LIN {X 0,Y 306.1,Z 708.373,A -85,B 0,C 180,E1 -15814.137,E2 -15814.137} C_VEL
LIN {X 0,Y 305.389,Z 716.212,A -85,B 0,C 180,E1 -15815.891,E2 -15815.891} C_VEL
LIN {X 0,Y 304.781,Z 723.046,A -85,B 0,C 180,E1 -15817.778,E2 -15817.778} C_VEL
LIN {X 0,Y 304.281,Z 728.72,A -85,B 0,C 180,E1 -15819.73,E2 -15819.73} C_VEL
LIN {X 0,Y 303.968,Z 733.701,A -85,B 0,C 180,E1 -15821.947,E2 -15821.947} C_VEL
LIN {X 0,Y 303.7,Z 736.898,A -85,B 0,C 180,E1 -15823.878,E2 -15823.878} C_VEL
LIN {X 0,Y 303.693,Z 738.582,A -85,B 0,C 180,E1 -15825.253,E2 -15825.253} C_VEL
LIN {X 0,Y 303.726,Z 739.763,A -85,B 0,C 180,E1 -15826.621,E2 -15826.621} C_VEL
LIN {X 0,Y 303.775,Z 740.52,A -85,B 0,C 180,E1 -15827.982,E2 -15827.982} C_VEL
LIN {X 0,Y 303.846,Z 740.805,A -85,B 0,C 180,E1 -15829.337,E2 -15829.337} C_VEL
LIN {X 0,Y 304.067,Z 740.63,A -85,B 0,C 180,E1 -15830.69,E2 -15830.69} C_VEL
LIN {X 0,Y 304.571,Z 739.433,A -85,B 0,C 180,E1 -15832.866,E2 -15832.866} C_VEL
LIN {X 0,Y 305.119,Z 737.5,A -85,B 0,C 180,E1 -15834.714,E2 -15834.714} C_VEL
LIN {X 0,Y 305.872,Z 734.444,A -85,B 0,C 180,E1 -15836.707,E2 -15836.707} C_VEL
LIN {X 0,Y 306.957,Z 730.272,A -85,B 0,C 180,E1 -15838.689,E2 -15838.689} C_VEL
LIN {X 0,Y 308.29,Z 724.889,A -85,B 0,C 180,E1 -15840.654,E2 -15840.654} C_VEL
LIN {X 0,Y 309.912,Z 718.102,A -85,B 0,C 180,E1 -15842.6,E2 -15842.6} C_VEL
LIN {X 0,Y 311.8,Z 709.706,A -85,B 0,C 180,E1 -15844.525,E2 -15844.525} C_VEL
LIN {X 0,Y 313.607,Z 701.139,A -85,B 0,C 180,E1 -15846.111,E2 -15846.111} C_VEL
LIN {X 0,Y 315.629,Z 690.583,A -85,B 0,C 180,E1 -15847.678,E2 -15847.678} C_VEL
LIN {X 0,Y 317.548,Z 678.795,A -85,B 0,C 180,E1 -15849.073,E2 -15849.073} C_VEL
LIN {X 0,Y 319.183,Z 667.151,A -85,B 0,C 180,E1 -15850.146,E2 -15850.146} C_VEL
LIN {X 0,Y 320.659,Z 654.294,A -85,B 0,C 180,E1 -15851.057,E2 -15851.057} C_VEL
LIN {X 0,Y 321.639,Z 641.719,A -85,B 0,C 180,E1 -15851.701,E2 -15851.701} C_VEL
LIN {X 0,Y 327.348,Z 557.799,A -85,B 0,C 180,E1 -15854.48,E2 -15854.48} C_VEL
LIN {X 0,Y 324.65,Z 543.648,A -85,B 0,C 180,E1 -15855.568,E2 -15855.568} C_VEL
LIN {X 0,Y 322.218,Z 533.831,A -85,B 0,C 180,E1 -15856.472,E2 -15856.472} C_VEL
LIN {X 0,Y 321.255,Z 531.249,A -85,B 0,C 180,E1 -15856.85,E2 -15856.85} C_VEL
LIN {X 0,Y 319.768,Z 522.812,A -85,B 0,C 180,E1 -15859.25,E2 -15859.25} C_VEL
LIN {X 0,Y 317.79,Z 515.127,A -85,B 0,C 180,E1 -15861.741,E2 -15861.741} C_VEL
LIN {X 0,Y 314.834,Z 506.328,A -85,B 0,C 180,E1 -15865.096,E2 -15865.096} C_VEL
LIN {X 0,Y 312.795,Z 501.239,A -85,B 0,C 180,E1 -15867.497,E2 -15867.497} C_VEL
LIN {X 0,Y 311.453,Z 498.267,A -85,B 0,C 180,E1 -15869.132,E2 -15869.132} C_VEL
LIN {X 0,Y 309.651,Z 494.731,A -85,B 0,C 180,E1 -15871.468,E2 -15871.468} C_VEL
LIN {X 0,Y 307.866,Z 490.948,A -85,B 0,C 180,E1 -15874.8,E2 -15874.8} C_VEL
LIN {X 0,Y 306.495,Z 489.331,A -85,B 0,C 180,E1 -15878.252,E2 -15878.252} C_VEL
LIN {X 0,Y 306.389,Z 489.148,A -85,B 0,C 180,E1 -15880.8,E2 -15880.8} C_VEL
LIN {X 0,Y 306.896,Z 489.969,A -85,B 0,C 180,E1 -15883.394,E2 -15883.394} C_VEL
LIN {X 0,Y 307.742,Z 490.943,A -85,B 0,C 180,E1 -15885.07,E2 -15885.07} C_VEL
LIN {X 0,Y 309.036,Z 492.803,A -85,B 0,C 180,E1 -15886.978,E2 -15886.978} C_VEL
LIN {X 0,Y 310.792,Z 495.708,A -85,B 0,C 180,E1 -15889.019,E2 -15889.019} C_VEL
LIN {X 0,Y 311.754,Z 500.683,A -85,B 0,C 180,E1 -15890.858,E2 -15890.858} C_VEL
LIN {X 0,Y 313.715,Z 508.861,A -85,B 0,C 180,E1 -15893.27,E2 -15893.27} C_VEL
LIN {X 0,Y 316.652,Z 519.821,A -85,B 0,C 180,E1 -15895.88,E2 -15895.88} C_VEL
LIN {X 0,Y 318.261,Z 525.565,A -85,B 0,C 180,E1 -15897.05,E2 -15897.05} C_VEL
LIN {X 0,Y 318.722,Z 528.436,A -85,B 0,C 180,E1 -15897.522,E2 -15897.522} C_VEL
LIN {X 0,Y 319.138,Z 540.824,A -85,B 0,C 180,E1 -15899.045,E2 -15899.045} C_VEL
LIN {X 0,Y 319.554,Z 549.759,A -85,B 0,C 180,E1 -15900.025,E2 -15900.025} C_VEL
LIN {X 0,Y 322.061,Z 568.33,A -85,B 0,C 180,E1 -15901.352,E2 -15901.352} C_VEL
LIN {X 0,Y 323.432,Z 583.449,A -85,B 0,C 180,E1 -15902.268,E2 -15902.268} C_VEL
LIN {X 0,Y 324.12,Z 604.294,A -85,B 0,C 180,E1 -15903.302,E2 -15903.302} C_VEL
LIN {X 0,Y 319.77,Z 671.023,A -85,B 0,C 180,E1 -15905.532,E2 -15905.532} C_VEL
LIN {X 0,Y 318.573,Z 683.595,A -85,B 0,C 180,E1 -15906.17,E2 -15906.17} C_VEL
LIN {X 0,Y 316.88,Z 695.874,A -85,B 0,C 180,E1 -15906.987,E2 -15906.987} C_VEL
LIN {X 0,Y 315.082,Z 707.84,A -85,B 0,C 180,E1 -15908.059,E2 -15908.059} C_VEL
LIN {X 0,Y 313.189,Z 718.84,A -85,B 0,C 180,E1 -15909.301,E2 -15909.301} C_VEL
LIN {X 0,Y 311.227,Z 728.95,A -85,B 0,C 180,E1 -15910.714,E2 -15910.714} C_VEL
LIN {X 0,Y 309.221,Z 739.018,A -85,B 0,C 180,E1 -15912.471,E2 -15912.471} C_VEL
LIN {X 0,Y 307.655,Z 746.638,A -85,B 0,C 180,E1 -15914.088,E2 -15914.088} C_VEL
LIN {X 0,Y 306.374,Z 754.172,A -85,B 0,C 180,E1 -15916.06,E2 -15916.06} C_VEL
LIN {X 0,Y 305.148,Z 760.218,A -85,B 0,C 180,E1 -15918.035,E2 -15918.035} C_VEL
LIN {X 0,Y 304.434,Z 765.005,A -85,B 0,C 180,E1 -15920.027,E2 -15920.027} C_VEL
LIN {X 0,Y 303.993,Z 768.688,A -85,B 0,C 180,E1 -15922.024,E2 -15922.024} C_VEL
LIN {X 0,Y 303.79,Z 771.447,A -85,B 0,C 180,E1 -15924.148,E2 -15924.148} C_VEL
LIN {X 0,Y 303.815,Z 772.957,A -85,B 0,C 180,E1 -15926.018,E2 -15926.018} C_VEL
LIN {X 0,Y 303.831,Z 773.479,A -85,B 0,C 180,E1 -15927.346,E2 -15927.346} C_VEL
LIN {X 0,Y 303.992,Z 773.588,A -85,B 0,C 180,E1 -15928.673,E2 -15928.673} C_VEL
LIN {X 0,Y 304.145,Z 773.257,A -85,B 0,C 180,E1 -15929.998,E2 -15929.998} C_VEL
LIN {X 0,Y 304.122,Z 772.422,A -85,B 0,C 180,E1 -15931.322,E2 -15931.322} C_VEL
LIN {X 0,Y 303.942,Z 771.129,A -85,B 0,C 180,E1 -15932.648,E2 -15932.648} C_VEL
LIN {X 0,Y 303.973,Z 768.306,A -85,B 0,C 180,E1 -15934.639,E2 -15934.639} C_VEL
LIN {X 0,Y 303.973,Z 764.316,A -85,B 0,C 180,E1 -15936.636,E2 -15936.636} C_VEL
LIN {X 0,Y 304.177,Z 758.011,A -85,B 0,C 180,E1 -15938.97,E2 -15938.97} C_VEL
LIN {X 0,Y 304.53,Z 751.01,A -85,B 0,C 180,E1 -15940.973,E2 -15940.973} C_VEL
LIN {X 0,Y 305.136,Z 743.832,A -85,B 0,C 180,E1 -15942.637,E2 -15942.637} C_VEL
LIN {X 0,Y 305.93,Z 735.098,A -85,B 0,C 180,E1 -15944.295,E2 -15944.295} C_VEL
LIN {X 0,Y 306.682,Z 725.782,A -85,B 0,C 180,E1 -15945.743,E2 -15945.743} C_VEL
LIN {X 0,Y 307.668,Z 715.031,A -85,B 0,C 180,E1 -15947.101,E2 -15947.101} C_VEL
LIN {X 0,Y 308.706,Z 703.671,A -85,B 0,C 180,E1 -15948.24,E2 -15948.24} C_VEL
LIN {X 0,Y 309.621,Z 692.085,A -85,B 0,C 180,E1 -15949.214,E2 -15949.214} C_VEL
LIN {X 0,Y 310.951,Z 680.136,A -85,B 0,C 180,E1 -15950.246,E2 -15950.246} C_VEL
LIN {X 0,Y 312.033,Z 666.967,A -85,B 0,C 180,E1 -15951.077,E2 -15951.077} C_VEL
LIN {X 0,Y 312.717,Z 653.939,A -85,B 0,C 180,E1 -15951.634,E2 -15951.634} C_VEL
LIN {X 0,Y 313.765,Z 602.785,A -85,B 0,C 180,E1 -15952.834,E2 -15952.834} C_VEL
LIN {X 0,Y 308.483,Z 544.585,A -85,B 0,C 180,E1 -15954.582,E2 -15954.582} C_VEL
LIN {X 0,Y 308.397,Z 541.255,A -85,B 0,C 180,E1 -15954.824,E2 -15954.824} C_VEL
LIN {X 0,Y 310.949,Z 518.833,A -85,B 0,C 180,E1 -15959.442,E2 -15959.442} C_VEL
LIN {X 0,Y 311.402,Z 514.116,A -85,B 0,C 180,E1 -15960.424,E2 -15960.424} C_VEL
LIN {X 0,Y 309.178,Z 502.702,A -85,B 0,C 180,E1 -15963.059,E2 -15963.059} C_VEL
LIN {X 0,Y 305.98,Z 488.559,A -85,B 0,C 180,E1 -15966.494,E2 -15966.494} C_VEL
LIN {X 0,Y 305.482,Z 486.515,A -85,B 0,C 180,E1 -15967.096,E2 -15967.096} C_VEL
LIN {X 0,Y 305.402,Z 486.441,A -85,B 0,C 180,E1 -15970.587,E2 -15970.587} C_VEL
LIN {X 0,Y 305.414,Z 486.439,A -85,B 0,C 180,E1 -15973.654,E2 -15973.654} C_VEL
LIN {X 0,Y 305.445,Z 486.435,A -85,B 0,C 180,E1 -15977.412,E2 -15977.412} C_VEL
LIN {X 0,Y 305.448,Z 486.437,A -85,B 0,C 180,E1 -15979.89,E2 -15979.89} C_VEL
LIN {X 0,Y 305.453,Z 486.435,A -85,B 0,C 180,E1 -15983.634,E2 -15983.634} C_VEL
LIN {X 0,Y 305.455,Z 486.436,A -85,B 0,C 180,E1 -15986.481,E2 -15986.481} C_VEL
LIN {X 0,Y 305.452,Z 486.434,A -85,B 0,C 180,E1 -15989.589,E2 -15989.589} C_VEL
LIN {X 0,Y 305.505,Z 486.426,A -85,B 0,C 180,E1 -15992.606,E2 -15992.606} C_VEL
LIN {X 0,Y 305.496,Z 486.428,A -85,B 0,C 180,E1 -15995.537,E2 -15995.537} C_VEL
LIN {X 0,Y 305.507,Z 486.424,A -85,B 0,C 180,E1 -15999.814,E2 -15999.814} C_VEL
LIN {X 0,Y 305.562,Z 486.424,A -85,B 0,C 180,E1 -16002.602,E2 -16002.602} C_VEL
LIN {X 0,Y 305.636,Z 486.41,A -85,B 0,C 180,E1 -16005.348,E2 -16005.348} C_VEL
LIN {X 0,Y 305.625,Z 486.405,A -85,B 0,C 180,E1 -16009.399,E2 -16009.399} C_VEL
LIN {X 0,Y 305.799,Z 486.39,A -85,B 0,C 180,E1 -16012.073,E2 -16012.073} C_VEL
LIN {X 0,Y 305.674,Z 486.408,A -85,B 0,C 180,E1 -16014.723,E2 -16014.723} C_VEL
LIN {X 0,Y 305.943,Z 486.368,A -85,B 0,C 180,E1 -16018.683,E2 -16018.683} C_VEL
LIN {X 0,Y 305.945,Z 486.37,A -85,B 0,C 180,E1 -16021.316,E2 -16021.316} C_VEL
LIN {X 0,Y 305.837,Z 486.386,A -85,B 0,C 180,E1 -16026.597,E2 -16026.597} C_VEL
LIN {X 0,Y 305.722,Z 486.393,A -85,B 0,C 180,E1 -16029.26,E2 -16029.26} C_VEL
LIN {X 0,Y 305.575,Z 486.419,A -85,B 0,C 180,E1 -16033.296,E2 -16033.296} C_VEL
LIN {X 0,Y 305.58,Z 486.418,A -85,B 0,C 180,E1 -16036.02,E2 -16036.02} C_VEL
LIN {X 0,Y 305.563,Z 486.412,A -85,B 0,C 180,E1 -16039.445,E2 -16039.445} C_VEL
LIN {X 0,Y 305.477,Z 486.433,A -85,B 0,C 180,E1 -16043.042,E2 -16043.042} C_VEL
LIN {X 0,Y 305.54,Z 486.423,A -85,B 0,C 180,E1 -16046.23,E2 -16046.23} C_VEL
LIN {X 0,Y 305.482,Z 486.427,A -85,B 0,C 180,E1 -16049.051,E2 -16049.051} C_VEL
LIN {X 0,Y 305.452,Z 486.434,A -85,B 0,C 180,E1 -16053.518,E2 -16053.518} C_VEL
LIN {X 0,Y 305.46,Z 486.432,A -85,B 0,C 180,E1 -16056.741,E2 -16056.741} C_VEL
LIN {X 0,Y 305.443,Z 486.437,A -85,B 0,C 180,E1 -16060.601,E2 -16060.601} C_VEL
LIN {X 0,Y 305.45,Z 486.433,A -85,B 0,C 180,E1 -16064.502,E2 -16064.502} C_VEL
LIN {X 0,Y 305.485,Z 486.43,A -85,B 0,C 180,E1 -16068.154,E2 -16068.154} C_VEL
LIN {X 0,Y 305.512,Z 486.419,A -85,B 0,C 180,E1 -16071.606,E2 -16071.606} C_VEL
LIN {X 0,Y 305.454,Z 486.425,A -85,B 0,C 180,E1 -16074.889,E2 -16074.889} C_VEL
LIN {X 0,Y 305.443,Z 486.436,A -85,B 0,C 180,E1 -16078.357,E2 -16078.357} C_VEL
LIN {X 0,Y 305.512,Z 486.422,A -85,B 0,C 180,E1 -16081.116,E2 -16081.116} C_VEL
LIN {X 0,Y 305.564,Z 486.418,A -85,B 0,C 180,E1 -16084.09,E2 -16084.09} C_VEL
LIN {X 0,Y 305.494,Z 486.424,A -85,B 0,C 180,E1 -16088.405,E2 -16088.405} C_VEL
LIN {X 0,Y 305.584,Z 486.422,A -85,B 0,C 180,E1 -16091.22,E2 -16091.22} C_VEL
LIN {X 0,Y 305.644,Z 486.411,A -85,B 0,C 180,E1 -16095.351,E2 -16095.351} C_VEL
LIN {X 0,Y 305.707,Z 486.553,A -85,B 0,C 180,E1 -16099.932,E2 -16099.932} C_VEL
LIN {X 0,Y 305.883,Z 487.388,A -85,B 0,C 180,E1 -16100.15,E2 -16100.15} C_VEL
LIN {X 0,Y 312.598,Z 503.956,A -85,B 0,C 180,E1 -16101.041,E2 -16101.041} C_VEL
LIN {X 0,Y 314.88,Z 510.634,A -85,B 0,C 180,E1 -16101.35,E2 -16101.35} C_VEL
LIN {X 0,Y 314.07,Z 560.457,A -85,B 0,C 180,E1 -16102.492,E2 -16102.492} C_VEL
LIN {X 0,Y 313.952,Z 574.677,A -85,B 0,C 180,E1 -16102.924,E2 -16102.924} C_VEL
LIN {X 0,Y 313.664,Z 587.236,A -85,B 0,C 180,E1 -16103.57,E2 -16103.57} C_VEL
LIN {X 0,Y 313.042,Z 600.404,A -85,B 0,C 180,E1 -16104.527,E2 -16104.527} C_VEL
LIN {X 0,Y 312.25,Z 611.94,A -85,B 0,C 180,E1 -16105.646,E2 -16105.646} C_VEL
LIN {X 0,Y 311.224,Z 623.522,A -85,B 0,C 180,E1 -16107.09,E2 -16107.09} C_VEL
LIN {X 0,Y 310.181,Z 633.83,A -85,B 0,C 180,E1 -16108.704,E2 -16108.704} C_VEL
LIN {X 0,Y 309.233,Z 642.046,A -85,B 0,C 180,E1 -16110.295,E2 -16110.295} C_VEL
LIN {X 0,Y 308.234,Z 650.371,A -85,B 0,C 180,E1 -16112.289,E2 -16112.289} C_VEL
LIN {X 0,Y 307.512,Z 655.974,A -85,B 0,C 180,E1 -16113.934,E2 -16113.934} C_VEL
LIN {X 0,Y 306.855,Z 661.444,A -85,B 0,C 180,E1 -16115.918,E2 -16115.918} C_VEL
LIN {X 0,Y 306.38,Z 665.742,A -85,B 0,C 180,E1 -16117.913,E2 -16117.913} C_VEL
LIN {X 0,Y 306.11,Z 668.041,A -85,B 0,C 180,E1 -16119.25,E2 -16119.25} C_VEL
LIN {X 0,Y 305.904,Z 669.873,A -85,B 0,C 180,E1 -16120.593,E2 -16120.593} C_VEL
LIN {X 0,Y 305.83,Z 671.259,A -85,B 0,C 180,E1 -16121.938,E2 -16121.938} C_VEL
LIN {X 0,Y 305.794,Z 672.259,A -85,B 0,C 180,E1 -16123.289,E2 -16123.289} C_VEL
LIN {X 0,Y 305.972,Z 672.956,A -85,B 0,C 180,E1 -16125.268,E2 -16125.268} C_VEL
LIN {X 0,Y 306.299,Z 672.761,A -85,B 0,C 180,E1 -16127.357,E2 -16127.357} C_VEL
LIN {X 0,Y 306.603,Z 672.129,A -85,B 0,C 180,E1 -16128.72,E2 -16128.72} C_VEL
LIN {X 0,Y 307.084,Z 670.895,A -85,B 0,C 180,E1 -16130.228,E2 -16130.228} C_VEL
LIN {X 0,Y 308.179,Z 667.551,A -85,B 0,C 180,E1 -16132.813,E2 -16132.813} C_VEL
LIN {X 0,Y 309.356,Z 663.459,A -85,B 0,C 180,E1 -16134.952,E2 -16134.952} C_VEL
LIN {X 0,Y 310.922,Z 657.501,A -85,B 0,C 180,E1 -16137.243,E2 -16137.243} C_VEL
LIN {X 0,Y 312.567,Z 650.633,A -85,B 0,C 180,E1 -16139.287,E2 -16139.287} C_VEL
LIN {X 0,Y 314.093,Z 643.567,A -85,B 0,C 180,E1 -16140.975,E2 -16140.975} C_VEL
LIN {X 0,Y 315.828,Z 634.861,A -85,B 0,C 180,E1 -16142.66,E2 -16142.66} C_VEL
LIN {X 0,Y 317.415,Z 625.121,A -85,B 0,C 180,E1 -16144.185,E2 -16144.185} C_VEL
LIN {X 0,Y 319.053,Z 614.168,A -85,B 0,C 180,E1 -16145.545,E2 -16145.545} C_VEL
LIN {X 0,Y 320.382,Z 602.187,A -85,B 0,C 180,E1 -16146.712,E2 -16146.712} C_VEL
LIN {X 0,Y 321.249,Z 590.535,A -85,B 0,C 180,E1 -16147.579,E2 -16147.579} C_VEL
LIN {X 0,Y 321.812,Z 577.18,A -85,B 0,C 180,E1 -16148.297,E2 -16148.297} C_VEL
LIN {X 0,Y 322.017,Z 564.33,A -85,B 0,C 180,E1 -16148.718,E2 -16148.718} C_VEL
LIN {X 0,Y 322.867,Z 524.411,A -85,B 0,C 180,E1 -16149.652,E2 -16149.652} C_VEL
LIN {X 0,Y 322.78,Z 519.432,A -85,B 0,C 180,E1 -16149.79,E2 -16149.79} C_VEL
LIN {X 0,Y 314.618,Z 503.331,A -85,B 0,C 180,E1 -16151.126,E2 -16151.126} C_VEL
LIN {X 0,Y 306.886,Z 489.869,A -85,B 0,C 180,E1 -16152.436,E2 -16152.436} C_VEL
LIN {X 0,Y 305.572,Z 487.133,A -85,B 0,C 180,E1 -16152.76,E2 -16152.76} C_VEL
LIN {X 0,Y 305.436,Z 486.512,A -85,B 0,C 180,E1 -16153.069,E2 -16153.069} C_VEL
LIN {X 0,Y 305.48,Z 486.649,A -85,B 0,C 180,E1 -16154.78,E2 -16154.78} C_VEL
LIN {X 0,Y 308.996,Z 501.481,A -85,B 0,C 180,E1 -16158.127,E2 -16158.127} C_VEL
LIN {X 0,Y 309.183,Z 505.467,A -85,B 0,C 180,E1 -16158.939,E2 -16158.939} C_VEL
LIN {X 0,Y 308.31,Z 509.616,A -85,B 0,C 180,E1 -16159.712,E2 -16159.712} C_VEL
LIN {X 0,Y 304.494,Z 520.955,A -85,B 0,C 180,E1 -16161.743,E2 -16161.743} C_VEL
LIN {X 0,Y 303.995,Z 523.76,A -85,B 0,C 180,E1 -16162.284,E2 -16162.284} C_VEL
LIN {X 0,Y 303.84,Z 526.593,A -85,B 0,C 180,E1 -16162.776,E2 -16162.776} C_VEL
LIN {X 0,Y 307.352,Z 552.339,A -85,B 0,C 180,E1 -16163.82,E2 -16163.82} C_VEL
LIN {X 0,Y 304.452,Z 638.058,A -85,B 0,C 180,E1 -16166.457,E2 -16166.457} C_VEL
LIN {X 0,Y 303.842,Z 650.589,A -85,B 0,C 180,E1 -16167.074,E2 -16167.074} C_VEL
LIN {X 0,Y 302.95,Z 664.348,A -85,B 0,C 180,E1 -16168.048,E2 -16168.048} C_VEL
LIN {X 0,Y 302.061,Z 676.658,A -85,B 0,C 180,E1 -16169.212,E2 -16169.212} C_VEL
LIN {X 0,Y 301.016,Z 688.488,A -85,B 0,C 180,E1 -16170.64,E2 -16170.64} C_VEL
LIN {X 0,Y 300.057,Z 698.06,A -85,B 0,C 180,E1 -16172.067,E2 -16172.067} C_VEL
LIN {X 0,Y 299.115,Z 707.825,A -85,B 0,C 180,E1 -16173.862,E2 -16173.862} C_VEL
LIN {X 0,Y 298.367,Z 715.818,A -85,B 0,C 180,E1 -16175.657,E2 -16175.657} C_VEL
LIN {X 0,Y 297.666,Z 723.515,A -85,B 0,C 180,E1 -16177.805,E2 -16177.805} C_VEL
LIN {X 0,Y 297.152,Z 729.538,A -85,B 0,C 180,E1 -16179.944,E2 -16179.944} C_VEL
LIN {X 0,Y 296.845,Z 734.178,A -85,B 0,C 180,E1 -16182.075,E2 -16182.075} C_VEL
LIN {X 0,Y 296.647,Z 736.553,A -85,B 0,C 180,E1 -16183.484,E2 -16183.484} C_VEL
LIN {X 0,Y 296.601,Z 738.417,A -85,B 0,C 180,E1 -16184.892,E2 -16184.892} C_VEL
LIN {X 0,Y 296.642,Z 739.824,A -85,B 0,C 180,E1 -16186.296,E2 -16186.296} C_VEL
LIN {X 0,Y 296.66,Z 740.718,A -85,B 0,C 180,E1 -16187.69,E2 -16187.69} C_VEL
LIN {X 0,Y 296.733,Z 741.185,A -85,B 0,C 180,E1 -16189.078,E2 -16189.078} C_VEL
LIN {X 0,Y 296.951,Z 741.217,A -85,B 0,C 180,E1 -16190.464,E2 -16190.464} C_VEL
LIN {X 0,Y 297.491,Z 740.172,A -85,B 0,C 180,E1 -16192.861,E2 -16192.861} C_VEL
LIN {X 0,Y 298.017,Z 738.625,A -85,B 0,C 180,E1 -16194.588,E2 -16194.588} C_VEL
LIN {X 0,Y 298.809,Z 735.834,A -85,B 0,C 180,E1 -16196.63,E2 -16196.63} C_VEL
LIN {X 0,Y 299.903,Z 731.949,A -85,B 0,C 180,E1 -16198.658,E2 -16198.658} C_VEL
LIN {X 0,Y 301.275,Z 726.891,A -85,B 0,C 180,E1 -16200.669,E2 -16200.669} C_VEL
LIN {X 0,Y 302.933,Z 720.532,A -85,B 0,C 180,E1 -16202.66,E2 -16202.66} C_VEL
LIN {X 0,Y 304.896,Z 712.63,A -85,B 0,C 180,E1 -16204.628,E2 -16204.628} C_VEL
LIN {X 0,Y 306.771,Z 704.52,A -85,B 0,C 180,E1 -16206.248,E2 -16206.248} C_VEL
LIN {X 0,Y 309.024,Z 693.617,A -85,B 0,C 180,E1 -16208.008,E2 -16208.008} C_VEL
LIN {X 0,Y 311.051,Z 682.532,A -85,B 0,C 180,E1 -16209.429,E2 -16209.429} C_VEL
LIN {X 0,Y 313.023,Z 670.068,A -85,B 0,C 180,E1 -16210.675,E2 -16210.675} C_VEL
LIN {X 0,Y 314.644,Z 656.76,A -85,B 0,C 180,E1 -16211.679,E2 -16211.679} C_VEL
LIN {X 0,Y 315.807,Z 644.231,A -85,B 0,C 180,E1 -16212.369,E2 -16212.369} C_VEL
LIN {X 0,Y 317.967,Z 612.55,A -85,B 0,C 180,E1 -16213.485,E2 -16213.485} C_VEL
LIN {X 0,Y 321.987,Z 559.662,A -85,B 0,C 180,E1 -16215.266,E2 -16215.266} C_VEL
LIN {X 0,Y 319.744,Z 546.746,A -85,B 0,C 180,E1 -16216.296,E2 -16216.296} C_VEL
LIN {X 0,Y 317.543,Z 537.471,A -85,B 0,C 180,E1 -16217.18,E2 -16217.18} C_VEL
LIN {X 0,Y 315.11,Z 531.981,A -85,B 0,C 180,E1 -16218.027,E2 -16218.027} C_VEL
LIN {X 0,Y 313.657,Z 524.477,A -85,B 0,C 180,E1 -16220.322,E2 -16220.322} C_VEL
LIN {X 0,Y 311.977,Z 518.087,A -85,B 0,C 180,E1 -16222.535,E2 -16222.535} C_VEL
LIN {X 0,Y 309.618,Z 510.669,A -85,B 0,C 180,E1 -16225.549,E2 -16225.549} C_VEL
LIN {X 0,Y 307.249,Z 504.435,A -85,B 0,C 180,E1 -16228.709,E2 -16228.709} C_VEL
LIN {X 0,Y 305.209,Z 500.218,A -85,B 0,C 180,E1 -16231.568,E2 -16231.568} C_VEL
LIN {X 0,Y 304.116,Z 497.88,A -85,B 0,C 180,E1 -16233.698,E2 -16233.698} C_VEL
LIN {X 0,Y 303.198,Z 496.179,A -85,B 0,C 180,E1 -16235.775,E2 -16235.775} C_VEL
LIN {X 0,Y 302.59,Z 495.316,A -85,B 0,C 180,E1 -16237.841,E2 -16237.841} C_VEL
LIN {X 0,Y 302.586,Z 495.132,A -85,B 0,C 180,E1 -16240.568,E2 -16240.568} C_VEL
LIN {X 0,Y 302.874,Z 495.571,A -85,B 0,C 180,E1 -16242.294,E2 -16242.294} C_VEL
LIN {X 0,Y 303.586,Z 496.458,A -85,B 0,C 180,E1 -16244.137,E2 -16244.137} C_VEL
LIN {X 0,Y 304.889,Z 498.071,A -85,B 0,C 180,E1 -16246.246,E2 -16246.246} C_VEL
LIN {X 0,Y 306.375,Z 500.875,A -85,B 0,C 180,E1 -16248.297,E2 -16248.297} C_VEL
LIN {X 0,Y 307.103,Z 502.242,A -85,B 0,C 180,E1 -16249.043,E2 -16249.043} C_VEL
LIN {X 0,Y 307.963,Z 507.429,A -85,B 0,C 180,E1 -16250.888,E2 -16250.888} C_VEL
LIN {X 0,Y 309.631,Z 514.739,A -85,B 0,C 180,E1 -16253.02,E2 -16253.02} C_VEL
LIN {X 0,Y 312.643,Z 526.439,A -85,B 0,C 180,E1 -16255.805,E2 -16255.805} C_VEL
LIN {X 0,Y 313.659,Z 530.679,A -85,B 0,C 180,E1 -16256.647,E2 -16256.647} C_VEL
LIN {X 0,Y 313.893,Z 535.174,A -85,B 0,C 180,E1 -16257.282,E2 -16257.282} C_VEL
LIN {X 0,Y 314.176,Z 549.125,A -85,B 0,C 180,E1 -16258.955,E2 -16258.955} C_VEL
LIN {X 0,Y 316.494,Z 566.69,A -85,B 0,C 180,E1 -16260.297,E2 -16260.297} C_VEL
LIN {X 0,Y 317.86,Z 581.372,A -85,B 0,C 180,E1 -16261.271,E2 -16261.271} C_VEL
LIN {X 0,Y 318.529,Z 596.708,A -85,B 0,C 180,E1 -16262.098,E2 -16262.098} C_VEL
LIN {X 0,Y 318.573,Z 607.311,A -85,B 0,C 180,E1 -16262.595,E2 -16262.595} C_VEL
LIN {X 0,Y 313.995,Z 671.128,A -85,B 0,C 180,E1 -16264.786,E2 -16264.786} C_VEL
LIN {X 0,Y 312.596,Z 684.771,A -85,B 0,C 180,E1 -16265.508,E2 -16265.508} C_VEL
LIN {X 0,Y 310.477,Z 698.322,A -85,B 0,C 180,E1 -16266.485,E2 -16266.485} C_VEL
LIN {X 0,Y 308.63,Z 709.619,A -85,B 0,C 180,E1 -16267.576,E2 -16267.576} C_VEL
LIN {X 0,Y 306.169,Z 722.452,A -85,B 0,C 180,E1 -16269.156,E2 -16269.156} C_VEL
LIN {X 0,Y 303.973,Z 732.811,A -85,B 0,C 180,E1 -16270.761,E2 -16270.761} C_VEL
LIN {X 0,Y 301.947,Z 742.305,A -85,B 0,C 180,E1 -16272.613,E2 -16272.613} C_VEL
LIN {X 0,Y 300.356,Z 749.703,A -85,B 0,C 180,E1 -16274.388,E2 -16274.388} C_VEL
LIN {X 0,Y 298.995,Z 756.555,A -85,B 0,C 180,E1 -16276.403,E2 -16276.403} C_VEL
LIN {X 0,Y 297.929,Z 762.036,A -85,B 0,C 180,E1 -16278.431,E2 -16278.431} C_VEL
LIN {X 0,Y 297.224,Z 766.316,A -85,B 0,C 180,E1 -16280.47,E2 -16280.47} C_VEL
LIN {X 0,Y 296.921,Z 768.548,A -85,B 0,C 180,E1 -16281.833,E2 -16281.833} C_VEL
LIN {X 0,Y 296.705,Z 771.37,A -85,B 0,C 180,E1 -16284.185,E2 -16284.185} C_VEL
LIN {X 0,Y 296.72,Z 772.606,A -85,B 0,C 180,E1 -16285.923,E2 -16285.923} C_VEL
LIN {X 0,Y 296.746,Z 773.081,A -85,B 0,C 180,E1 -16287.283,E2 -16287.283} C_VEL
LIN {X 0,Y 296.897,Z 773.135,A -85,B 0,C 180,E1 -16288.641,E2 -16288.641} C_VEL
LIN {X 0,Y 297.084,Z 772.705,A -85,B 0,C 180,E1 -16289.998,E2 -16289.998} C_VEL
LIN {X 0,Y 297.04,Z 771.815,A -85,B 0,C 180,E1 -16291.353,E2 -16291.353} C_VEL
LIN {X 0,Y 296.858,Z 770.473,A -85,B 0,C 180,E1 -16292.712,E2 -16292.712} C_VEL
LIN {X 0,Y 296.905,Z 767.549,A -85,B 0,C 180,E1 -16294.75,E2 -16294.75} C_VEL
LIN {X 0,Y 296.912,Z 763.437,A -85,B 0,C 180,E1 -16296.795,E2 -16296.795} C_VEL
LIN {X 0,Y 297.138,Z 756.97,A -85,B 0,C 180,E1 -16299.184,E2 -16299.184} C_VEL
LIN {X 0,Y 297.517,Z 749.825,A -85,B 0,C 180,E1 -16301.235,E2 -16301.235} C_VEL
LIN {X 0,Y 298.253,Z 740.767,A -85,B 0,C 180,E1 -16303.28,E2 -16303.28} C_VEL
LIN {X 0,Y 299.126,Z 731.462,A -85,B 0,C 180,E1 -16304.975,E2 -16304.975} C_VEL
LIN {X 0,Y 300.085,Z 721.105,A -85,B 0,C 180,E1 -16306.495,E2 -16306.495} C_VEL
LIN {X 0,Y 301.202,Z 709.719,A -85,B 0,C 180,E1 -16307.831,E2 -16307.831} C_VEL
LIN {X 0,Y 302.196,Z 696.87,A -85,B 0,C 180,E1 -16308.999,E2 -16308.999} C_VEL
LIN {X 0,Y 303.969,Z 680.963,A -85,B 0,C 180,E1 -16310.466,E2 -16310.466} C_VEL
LIN {X 0,Y 305.125,Z 667.949,A -85,B 0,C 180,E1 -16311.357,E2 -16311.357} C_VEL
LIN {X 0,Y 305.882,Z 654.764,A -85,B 0,C 180,E1 -16311.964,E2 -16311.964} C_VEL
LIN {X 0,Y 306.403,Z 634.31,A -85,B 0,C 180,E1 -16312.5,E2 -16312.5} C_VEL
LIN {X 0,Y 306.902,Z 601.653,A -85,B 0,C 180,E1 -16313.265,E2 -16313.265} C_VEL
LIN {X 0,Y 301.6,Z 543.63,A -85,B 0,C 180,E1 -16315.037,E2 -16315.037} C_VEL
LIN {X 0,Y 301.511,Z 540.507,A -85,B 0,C 180,E1 -16315.26,E2 -16315.26} C_VEL
LIN {X 0,Y 304.073,Z 519.032,A -85,B 0,C 180,E1 -16319.794,E2 -16319.794} C_VEL
LIN {X 0,Y 304.363,Z 514.64,A -85,B 0,C 180,E1 -16320.743,E2 -16320.743} C_VEL
LIN {X 0,Y 301.259,Z 499.494,A -85,B 0,C 180,E1 -16324.358,E2 -16324.358} C_VEL
LIN {X 0,Y 298.438,Z 487.433,A -85,B 0,C 180,E1 -16327.464,E2 -16327.464} C_VEL
LIN {X 0,Y 298.34,Z 487.319,A -85,B 0,C 180,E1 -16331.266,E2 -16331.266} C_VEL
LIN {X 0,Y 298.346,Z 487.32,A -85,B 0,C 180,E1 -16335.033,E2 -16335.033} C_VEL
LIN {X 0,Y 298.374,Z 487.317,A -85,B 0,C 180,E1 -16338.736,E2 -16338.736} C_VEL
LIN {X 0,Y 298.386,Z 487.319,A -85,B 0,C 180,E1 -16342.237,E2 -16342.237} C_VEL
LIN {X 0,Y 298.397,Z 487.307,A -85,B 0,C 180,E1 -16345.579,E2 -16345.579} C_VEL
LIN {X 0,Y 298.385,Z 487.315,A -85,B 0,C 180,E1 -16348.789,E2 -16348.789} C_VEL
LIN {X 0,Y 298.449,Z 487.302,A -85,B 0,C 180,E1 -16351.902,E2 -16351.902} C_VEL
LIN {X 0,Y 298.471,Z 487.304,A -85,B 0,C 180,E1 -16354.922,E2 -16354.922} C_VEL
LIN {X 0,Y 298.438,Z 487.303,A -85,B 0,C 180,E1 -16359.314,E2 -16359.314} C_VEL
LIN {X 0,Y 298.525,Z 487.296,A -85,B 0,C 180,E1 -16362.178,E2 -16362.178} C_VEL
LIN {X 0,Y 298.581,Z 487.29,A -85,B 0,C 180,E1 -16364.994,E2 -16364.994} C_VEL
LIN {X 0,Y 298.58,Z 487.283,A -85,B 0,C 180,E1 -16369.146,E2 -16369.146} C_VEL
LIN {X 0,Y 298.745,Z 487.268,A -85,B 0,C 180,E1 -16371.885,E2 -16371.885} C_VEL
LIN {X 0,Y 298.645,Z 487.285,A -85,B 0,C 180,E1 -16374.598,E2 -16374.598} C_VEL
LIN {X 0,Y 298.91,Z 487.243,A -85,B 0,C 180,E1 -16378.652,E2 -16378.652} C_VEL
LIN {X 0,Y 298.912,Z 487.246,A -85,B 0,C 180,E1 -16381.347,E2 -16381.347} C_VEL
LIN {X 0,Y 298.783,Z 487.262,A -85,B 0,C 180,E1 -16386.754,E2 -16386.754} C_VEL
LIN {X 0,Y 298.667,Z 487.27,A -85,B 0,C 180,E1 -16389.48,E2 -16389.48} C_VEL
LIN {X 0,Y 298.538,Z 487.295,A -85,B 0,C 180,E1 -16393.615,E2 -16393.615} C_VEL
LIN {X 0,Y 298.535,Z 487.298,A -85,B 0,C 180,E1 -16396.409,E2 -16396.409} C_VEL
LIN {X 0,Y 298.498,Z 487.291,A -85,B 0,C 180,E1 -16399.655,E2 -16399.655} C_VEL
LIN {X 0,Y 298.444,Z 487.306,A -85,B 0,C 180,E1 -16403.598,E2 -16403.598} C_VEL
LIN {X 0,Y 298.478,Z 487.305,A -85,B 0,C 180,E1 -16406.575,E2 -16406.575} C_VEL
LIN {X 0,Y 298.408,Z 487.305,A -85,B 0,C 180,E1 -16409.642,E2 -16409.642} C_VEL
LIN {X 0,Y 298.382,Z 487.319,A -85,B 0,C 180,E1 -16412.801,E2 -16412.801} C_VEL
LIN {X 0,Y 298.432,Z 487.306,A -85,B 0,C 180,E1 -16416.808,E2 -16416.808} C_VEL
LIN {X 0,Y 298.376,Z 487.319,A -85,B 0,C 180,E1 -16421.089,E2 -16421.089} C_VEL
LIN {X 0,Y 298.405,Z 487.311,A -85,B 0,C 180,E1 -16424.955,E2 -16424.955} C_VEL
LIN {X 0,Y 298.444,Z 487.311,A -85,B 0,C 180,E1 -16428.752,E2 -16428.752} C_VEL
LIN {X 0,Y 298.44,Z 487.299,A -85,B 0,C 180,E1 -16432.249,E2 -16432.249} C_VEL
LIN {X 0,Y 298.4,Z 487.309,A -85,B 0,C 180,E1 -16435.583,E2 -16435.583} C_VEL
LIN {X 0,Y 298.387,Z 487.318,A -85,B 0,C 180,E1 -16438.793,E2 -16438.793} C_VEL
LIN {X 0,Y 298.455,Z 487.295,A -85,B 0,C 180,E1 -16441.906,E2 -16441.906} C_VEL
LIN {X 0,Y 298.478,Z 487.305,A -85,B 0,C 180,E1 -16444.926,E2 -16444.926} C_VEL
LIN {X 0,Y 298.443,Z 487.307,A -85,B 0,C 180,E1 -16449.317,E2 -16449.317} C_VEL
LIN {X 0,Y 298.532,Z 487.296,A -85,B 0,C 180,E1 -16452.182,E2 -16452.182} C_VEL
LIN {X 0,Y 298.589,Z 487.294,A -85,B 0,C 180,E1 -16454.997,E2 -16454.997} C_VEL
LIN {X 0,Y 298.636,Z 487.473,A -85,B 0,C 180,E1 -16459.459,E2 -16459.459} C_VEL
LIN {X 0,Y 298.913,Z 488.637,A -85,B 0,C 180,E1 -16459.697,E2 -16459.697} C_VEL
LIN {X 0,Y 305.57,Z 504.686,A -85,B 0,C 180,E1 -16460.586,E2 -16460.586} C_VEL
LIN {X 0,Y 308.193,Z 512.453,A -85,B 0,C 180,E1 -16460.956,E2 -16460.956} C_VEL
LIN {X 0,Y 307.342,Z 560.405,A -85,B 0,C 180,E1 -16462.076,E2 -16462.076} C_VEL
LIN {X 0,Y 307.255,Z 574.132,A -85,B 0,C 180,E1 -16462.486,E2 -16462.486} C_VEL
LIN {X 0,Y 307.019,Z 586.547,A -85,B 0,C 180,E1 -16463.1,E2 -16463.1} C_VEL
LIN {X 0,Y 306.477,Z 598.167,A -85,B 0,C 180,E1 -16463.914,E2 -16463.914} C_VEL
LIN {X 0,Y 305.644,Z 610.423,A -85,B 0,C 180,E1 -16465.056,E2 -16465.056} C_VEL
LIN {X 0,Y 304.709,Z 621.394,A -85,B 0,C 180,E1 -16466.366,E2 -16466.366} C_VEL
LIN {X 0,Y 303.758,Z 630.32,A -85,B 0,C 180,E1 -16467.682,E2 -16467.682} C_VEL
LIN {X 0,Y 302.681,Z 639.885,A -85,B 0,C 180,E1 -16469.421,E2 -16469.421} C_VEL
LIN {X 0,Y 301.613,Z 648.399,A -85,B 0,C 180,E1 -16471.337,E2 -16471.337} C_VEL
LIN {X 0,Y 300.743,Z 655.587,A -85,B 0,C 180,E1 -16473.351,E2 -16473.351} C_VEL
LIN {X 0,Y 299.988,Z 661.352,A -85,B 0,C 180,E1 -16475.379,E2 -16475.379} C_VEL
LIN {X 0,Y 299.453,Z 665.894,A -85,B 0,C 180,E1 -16477.419,E2 -16477.419} C_VEL
LIN {X 0,Y 299.023,Z 669.376,A -85,B 0,C 180,E1 -16479.472,E2 -16479.472} C_VEL
LIN {X 0,Y 298.846,Z 671.116,A -85,B 0,C 180,E1 -16480.846,E2 -16480.846} C_VEL
LIN {X 0,Y 298.788,Z 672.449,A -85,B 0,C 180,E1 -16482.224,E2 -16482.224} C_VEL
LIN {X 0,Y 298.779,Z 673.393,A -85,B 0,C 180,E1 -16483.607,E2 -16483.607} C_VEL
LIN {X 0,Y 298.973,Z 673.959,A -85,B 0,C 180,E1 -16485.467,E2 -16485.467} C_VEL
LIN {X 0,Y 299.36,Z 673.685,A -85,B 0,C 180,E1 -16487.772,E2 -16487.772} C_VEL
LIN {X 0,Y 299.71,Z 672.972,A -85,B 0,C 180,E1 -16489.167,E2 -16489.167} C_VEL
LIN {X 0,Y 300.187,Z 671.8,A -85,B 0,C 180,E1 -16490.562,E2 -16490.562} C_VEL
LIN {X 0,Y 301.102,Z 669.235,A -85,B 0,C 180,E1 -16492.654,E2 -16492.654} C_VEL
LIN {X 0,Y 302.361,Z 665.128,A -85,B 0,C 180,E1 -16494.974,E2 -16494.974} C_VEL
LIN {X 0,Y 303.604,Z 660.736,A -85,B 0,C 180,E1 -16496.836,E2 -16496.836} C_VEL
LIN {X 0,Y 305.306,Z 654.282,A -85,B 0,C 180,E1 -16498.987,E2 -16498.987} C_VEL
LIN {X 0,Y 307.08,Z 646.574,A -85,B 0,C 180,E1 -16500.996,E2 -16500.996} C_VEL
LIN {X 0,Y 309.045,Z 637.607,A -85,B 0,C 180,E1 -16502.846,E2 -16502.846} C_VEL
LIN {X 0,Y 310.72,Z 628.119,A -85,B 0,C 180,E1 -16504.437,E2 -16504.437} C_VEL
LIN {X 0,Y 312.378,Z 617.816,A -85,B 0,C 180,E1 -16505.802,E2 -16505.802} C_VEL
LIN {X 0,Y 313.828,Z 606.395,A -85,B 0,C 180,E1 -16507.005,E2 -16507.005} C_VEL
LIN {X 0,Y 314.837,Z 594.631,A -85,B 0,C 180,E1 -16507.974,E2 -16507.974} C_VEL
LIN {X 0,Y 315.601,Z 581.548,A -85,B 0,C 180,E1 -16508.744,E2 -16508.744} C_VEL
LIN {X 0,Y 315.855,Z 569.208,A -85,B 0,C 180,E1 -16509.23,E2 -16509.23} C_VEL
LIN {X 0,Y 316.535,Z 532.323,A -85,B 0,C 180,E1 -16510.136,E2 -16510.136} C_VEL
LIN {X 0,Y 316.833,Z 521.992,A -85,B 0,C 180,E1 -16510.376,E2 -16510.376} C_VEL
LIN {X 0,Y 309.261,Z 507.042,A -85,B 0,C 180,E1 -16511.663,E2 -16511.663} C_VEL
LIN {X 0,Y 300.296,Z 491.368,A -85,B 0,C 180,E1 -16513.245,E2 -16513.245} C_VEL
LIN {X 0,Y 298.644,Z 488.493,A -85,B 0,C 180,E1 -16513.582,E2 -16513.582} C_VEL
LIN {X 0,Y 298.4,Z 487.445,A -85,B 0,C 180,E1 -16513.897,E2 -16513.897} C_VEL
LIN {X 0,Y 298.433,Z 487.647,A -85,B 0,C 180,E1 -16514.42,E2 -16514.42} C_VEL
LIN {X 0,Y 302.276,Z 503.706,A -85,B 0,C 180,E1 -16518.077,E2 -16518.077} C_VEL
LIN {X 0,Y 304.549,Z 515.299,A -85,B 0,C 180,E1 -16520.61,E2 -16520.61} C_VEL
LIN {X 0,Y 303.995,Z 523.76,A -85,B 0,C 180,E1 -16522.284,E2 -16522.284} C_VEL
LIN {X 0,Y 303.149,Z 526.055,A -85,B 0,C 180,E1 -16522.569,E2 -16522.569} C_VEL
LIN {X 0,Y 301.567,Z 528.556,A -85,B 0,C 180,E1 -16522.683,E2 -16522.683} C_VEL
LIN {X 0,Y 297.643,Z 534.86,A -85,B 0,C 180,E1 -16522.707,E2 -16522.707} C_VEL
LIN {X 0,Y 296.629,Z 538.446,A -85,B 0,C 180,E1 -16522.769,E2 -16522.769} C_VEL
LIN {X 0,Y 296.954,Z 542.135,A -85,B 0,C 180,E1 -16522.893,E2 -16522.893} C_VEL
LIN {X 0,Y 300.262,Z 552.273,A -85,B 0,C 180,E1 -16523.434,E2 -16523.434} C_VEL
LIN {X 0,Y 300.447,Z 554.417,A -85,B 0,C 180,E1 -16523.518,E2 -16523.518} C_VEL
LIN {X 0,Y 297.458,Z 639.014,A -85,B 0,C 180,E1 -16526.223,E2 -16526.223} C_VEL
LIN {X 0,Y 296.797,Z 651.958,A -85,B 0,C 180,E1 -16526.9,E2 -16526.9} C_VEL
LIN {X 0,Y 295.911,Z 665.5,A -85,B 0,C 180,E1 -16527.9,E2 -16527.9} C_VEL
LIN {X 0,Y 295.016,Z 677.277,A -85,B 0,C 180,E1 -16529.053,E2 -16529.053} C_VEL
LIN {X 0,Y 293.981,Z 688.662,A -85,B 0,C 180,E1 -16530.458,E2 -16530.458} C_VEL
LIN {X 0,Y 292.929,Z 699.365,A -85,B 0,C 180,E1 -16532.107,E2 -16532.107} C_VEL
LIN {X 0,Y 291.948,Z 708.982,A -85,B 0,C 180,E1 -16533.94,E2 -16533.94} C_VEL
LIN {X 0,Y 291.231,Z 716.875,A -85,B 0,C 180,E1 -16535.78,E2 -16535.78} C_VEL
LIN {X 0,Y 290.518,Z 724.419,A -85,B 0,C 180,E1 -16537.978,E2 -16537.978} C_VEL
LIN {X 0,Y 290.025,Z 730.366,A -85,B 0,C 180,E1 -16540.169,E2 -16540.169} C_VEL
LIN {X 0,Y 289.713,Z 734.917,A -85,B 0,C 180,E1 -16542.349,E2 -16542.349} C_VEL
LIN {X 0,Y 289.521,Z 738.204,A -85,B 0,C 180,E1 -16544.514,E2 -16544.514} C_VEL
LIN {X 0,Y 289.537,Z 739.942,A -85,B 0,C 180,E1 -16546.158,E2 -16546.158} C_VEL
LIN {X 0,Y 289.55,Z 740.865,A -85,B 0,C 180,E1 -16547.383,E2 -16547.383} C_VEL
LIN {X 0,Y 289.617,Z 741.512,A -85,B 0,C 180,E1 -16548.807,E2 -16548.807} C_VEL
LIN {X 0,Y 289.835,Z 741.692,A -85,B 0,C 180,E1 -16550.228,E2 -16550.228} C_VEL
LIN {X 0,Y 290.418,Z 740.907,A -85,B 0,C 180,E1 -16552.846,E2 -16552.846} C_VEL
LIN {X 0,Y 290.919,Z 739.629,A -85,B 0,C 180,E1 -16554.455,E2 -16554.455} C_VEL
LIN {X 0,Y 291.706,Z 737.12,A -85,B 0,C 180,E1 -16556.547,E2 -16556.547} C_VEL
LIN {X 0,Y 292.841,Z 733.565,A -85,B 0,C 180,E1 -16558.625,E2 -16558.625} C_VEL
LIN {X 0,Y 294.248,Z 728.867,A -85,B 0,C 180,E1 -16560.685,E2 -16560.685} C_VEL
LIN {X 0,Y 295.944,Z 722.897,A -85,B 0,C 180,E1 -16562.723,E2 -16562.723} C_VEL
LIN {X 0,Y 297.98,Z 715.401,A -85,B 0,C 180,E1 -16564.736,E2 -16564.736} C_VEL
LIN {X 0,Y 300.316,Z 706.166,A -85,B 0,C 180,E1 -16566.72,E2 -16566.72} C_VEL
LIN {X 0,Y 302.477,Z 696.648,A -85,B 0,C 180,E1 -16568.35,E2 -16568.35} C_VEL
LIN {X 0,Y 304.834,Z 684.84,A -85,B 0,C 180,E1 -16569.958,E2 -16569.958} C_VEL
LIN {X 0,Y 306.876,Z 672.858,A -85,B 0,C 180,E1 -16571.226,E2 -16571.226} C_VEL
LIN {X 0,Y 308.635,Z 660.539,A -85,B 0,C 180,E1 -16572.243,E2 -16572.243} C_VEL
LIN {X 0,Y 310.067,Z 647.024,A -85,B 0,C 180,E1 -16573.059,E2 -16573.059} C_VEL
LIN {X 0,Y 311.21,Z 631.51,A -85,B 0,C 180,E1 -16573.685,E2 -16573.685} C_VEL
LIN {X 0,Y 316.801,Z 561.631,A -85,B 0,C 180,E1 -16576.094,E2 -16576.094} C_VEL
LIN {X 0,Y 315.324,Z 551.931,A -85,B 0,C 180,E1 -16576.865,E2 -16576.865} C_VEL
LIN {X 0,Y 313.053,Z 541.31,A -85,B 0,C 180,E1 -16577.896,E2 -16577.896} C_VEL
LIN {X 0,Y 309.07,Z 532.838,A -85,B 0,C 180,E1 -16579.304,E2 -16579.304} C_VEL
LIN {X 0,Y 307.466,Z 525.176,A -85,B 0,C 180,E1 -16581.85,E2 -16581.85} C_VEL
LIN {X 0,Y 305.054,Z 516.803,A -85,B 0,C 180,E1 -16585.229,E2 -16585.229} C_VEL
LIN {X 0,Y 302.991,Z 510.92,A -85,B 0,C 180,E1 -16588.181,E2 -16588.181} C_VEL
LIN {X 0,Y 301.312,Z 506.85,A -85,B 0,C 180,E1 -16590.874,E2 -16590.874} C_VEL
LIN {X 0,Y 299.469,Z 502.722,A -85,B 0,C 180,E1 -16594.773,E2 -16594.773} C_VEL
LIN {X 0,Y 298.811,Z 501.544,A -85,B 0,C 180,E1 -16596.898,E2 -16596.898} C_VEL
LIN {X 0,Y 298.661,Z 501.053,A -85,B 0,C 180,E1 -16599.447,E2 -16599.447} C_VEL
LIN {X 0,Y 298.824,Z 501.246,A -85,B 0,C 180,E1 -16601.188,E2 -16601.188} C_VEL
LIN {X 0,Y 299.396,Z 502.045,A -85,B 0,C 180,E1 -16603.304,E2 -16603.304} C_VEL
LIN {X 0,Y 301.272,Z 504.338,A -85,B 0,C 180,E1 -16606.317,E2 -16606.317} C_VEL
LIN {X 0,Y 302.542,Z 506.685,A -85,B 0,C 180,E1 -16608.019,E2 -16608.019} C_VEL
LIN {X 0,Y 303.213,Z 508.456,A -85,B 0,C 180,E1 -16608.929,E2 -16608.929} C_VEL
LIN {X 0,Y 304.364,Z 515.084,A -85,B 0,C 180,E1 -16611.187,E2 -16611.187} C_VEL
LIN {X 0,Y 306.14,Z 523.36,A -85,B 0,C 180,E1 -16613.465,E2 -16613.465} C_VEL
LIN {X 0,Y 308.524,Z 532.839,A -85,B 0,C 180,E1 -16615.666,E2 -16615.666} C_VEL
LIN {X 0,Y 308.988,Z 536.285,A -85,B 0,C 180,E1 -16616.275,E2 -16616.275} C_VEL
LIN {X 0,Y 308.964,Z 548.48,A -85,B 0,C 180,E1 -16617.809,E2 -16617.809} C_VEL
LIN {X 0,Y 311.023,Z 564.092,A -85,B 0,C 180,E1 -16619.117,E2 -16619.117} C_VEL
LIN {X 0,Y 312.641,Z 581.213,A -85,B 0,C 180,E1 -16620.324,E2 -16620.324} C_VEL
LIN {X 0,Y 313.219,Z 597.185,A -85,B 0,C 180,E1 -16621.239,E2 -16621.239} C_VEL
LIN {X 0,Y 313.16,Z 608.389,A -85,B 0,C 180,E1 -16621.78,E2 -16621.78} C_VEL
LIN {X 0,Y 308.457,Z 669.855,A -85,B 0,C 180,E1 -16623.938,E2 -16623.938} C_VEL
LIN {X 0,Y 306.918,Z 683.501,A -85,B 0,C 180,E1 -16624.662,E2 -16624.662} C_VEL
LIN {X 0,Y 304.738,Z 697.188,A -85,B 0,C 180,E1 -16625.652,E2 -16625.652} C_VEL
LIN {X 0,Y 302.755,Z 708.619,A -85,B 0,C 180,E1 -16626.755,E2 -16626.755} C_VEL
LIN {X 0,Y 300.383,Z 720.342,A -85,B 0,C 180,E1 -16628.194,E2 -16628.194} C_VEL
LIN {X 0,Y 298.238,Z 729.941,A -85,B 0,C 180,E1 -16629.658,E2 -16629.658} C_VEL
LIN {X 0,Y 296.184,Z 738.84,A -85,B 0,C 180,E1 -16631.315,E2 -16631.315} C_VEL
LIN {X 0,Y 294.061,Z 747.622,A -85,B 0,C 180,E1 -16633.331,E2 -16633.331} C_VEL
LIN {X 0,Y 292.62,Z 754.72,A -85,B 0,C 180,E1 -16635.391,E2 -16635.391} C_VEL
LIN {X 0,Y 291.219,Z 760.46,A -85,B 0,C 180,E1 -16637.453,E2 -16637.453} C_VEL
LIN {X 0,Y 290.411,Z 764.997,A -85,B 0,C 180,E1 -16639.541,E2 -16639.541} C_VEL
LIN {X 0,Y 289.871,Z 768.433,A -85,B 0,C 180,E1 -16641.633,E2 -16641.633} C_VEL
LIN {X 0,Y 289.67,Z 770.168,A -85,B 0,C 180,E1 -16643.03,E2 -16643.03} C_VEL
LIN {X 0,Y 289.608,Z 771.422,A -85,B 0,C 180,E1 -16644.427,E2 -16644.427} C_VEL
LIN {X 0,Y 289.63,Z 772.261,A -85,B 0,C 180,E1 -16645.823,E2 -16645.823} C_VEL
LIN {X 0,Y 289.663,Z 772.685,A -85,B 0,C 180,E1 -16647.216,E2 -16647.216} C_VEL
LIN {X 0,Y 289.805,Z 772.643,A -85,B 0,C 180,E1 -16648.608,E2 -16648.608} C_VEL
LIN {X 0,Y 290.024,Z 772.151,A -85,B 0,C 180,E1 -16649.998,E2 -16649.998} C_VEL
LIN {X 0,Y 289.961,Z 771.205,A -85,B 0,C 180,E1 -16651.387,E2 -16651.387} C_VEL
LIN {X 0,Y 289.778,Z 769.772,A -85,B 0,C 180,E1 -16652.778,E2 -16652.778} C_VEL
LIN {X 0,Y 289.838,Z 766.719,A -85,B 0,C 180,E1 -16654.866,E2 -16654.866} C_VEL
LIN {X 0,Y 289.848,Z 762.457,A -85,B 0,C 180,E1 -16656.961,E2 -16656.961} C_VEL
LIN {X 0,Y 290.034,Z 756.882,A -85,B 0,C 180,E1 -16659.06,E2 -16659.06} C_VEL
LIN {X 0,Y 290.423,Z 749.818,A -85,B 0,C 180,E1 -16661.16,E2 -16661.16} C_VEL
LIN {X 0,Y 291.03,Z 742.553,A -85,B 0,C 180,E1 -16662.905,E2 -16662.905} C_VEL
LIN {X 0,Y 291.879,Z 733.694,A -85,B 0,C 180,E1 -16664.642,E2 -16664.642} C_VEL
LIN {X 0,Y 292.675,Z 724.318,A -85,B 0,C 180,E1 -16666.152,E2 -16666.152} C_VEL
LIN {X 0,Y 293.742,Z 713.409,A -85,B 0,C 180,E1 -16667.579,E2 -16667.579} C_VEL
LIN {X 0,Y 294.783,Z 701.79,A -85,B 0,C 180,E1 -16668.773,E2 -16668.773} C_VEL
LIN {X 0,Y 295.462,Z 694.439,A -85,B 0,C 180,E1 -16669.449,E2 -16669.449} C_VEL
LIN {X 0,Y 296.883,Z 682.735,A -85,B 0,C 180,E1 -16670.615,E2 -16670.615} C_VEL
LIN {X 0,Y 298.083,Z 670.607,A -85,B 0,C 180,E1 -16671.523,E2 -16671.523} C_VEL
LIN {X 0,Y 298.902,Z 657.692,A -85,B 0,C 180,E1 -16672.218,E2 -16672.218} C_VEL
LIN {X 0,Y 299.432,Z 644.102,A -85,B 0,C 180,E1 -16672.665,E2 -16672.665} C_VEL
LIN {X 0,Y 300.141,Z 601.815,A -85,B 0,C 180,E1 -16673.676,E2 -16673.676} C_VEL
LIN {X 0,Y 294.636,Z 540.717,A -85,B 0,C 180,E1 -16675.613,E2 -16675.613} C_VEL
LIN {X 0,Y 294.688,Z 539.346,A -85,B 0,C 180,E1 -16675.798,E2 -16675.798} C_VEL
LIN {X 0,Y 297.204,Z 519.174,A -85,B 0,C 180,E1 -16680.163,E2 -16680.163} C_VEL
LIN {X 0,Y 297.395,Z 515.758,A -85,B 0,C 180,E1 -16680.927,E2 -16680.927} C_VEL
LIN {X 0,Y 294.331,Z 500.876,A -85,B 0,C 180,E1 -16684.58,E2 -16684.58} C_VEL
LIN {X 0,Y 291.374,Z 488.313,A -85,B 0,C 180,E1 -16687.899,E2 -16687.899} C_VEL
LIN {X 0,Y 291.287,Z 488.199,A -85,B 0,C 180,E1 -16691.586,E2 -16691.586} C_VEL
LIN {X 0,Y 291.282,Z 488.201,A -85,B 0,C 180,E1 -16695.596,E2 -16695.596} C_VEL
LIN {X 0,Y 291.321,Z 488.195,A -85,B 0,C 180,E1 -16699.355,E2 -16699.355} C_VEL
LIN {X 0,Y 291.38,Z 488.188,A -85,B 0,C 180,E1 -16702.915,E2 -16702.915} C_VEL
LIN {X 0,Y 291.334,Z 488.192,A -85,B 0,C 180,E1 -16706.3,E2 -16706.3} C_VEL
LIN {X 0,Y 291.376,Z 488.187,A -85,B 0,C 180,E1 -16710.259,E2 -16710.259} C_VEL
LIN {X 0,Y 291.401,Z 488.184,A -85,B 0,C 180,E1 -16714.27,E2 -16714.27} C_VEL
LIN {X 0,Y 291.37,Z 488.188,A -85,B 0,C 180,E1 -16717.298,E2 -16717.298} C_VEL
LIN {X 0,Y 291.446,Z 488.174,A -85,B 0,C 180,E1 -16720.269,E2 -16720.269} C_VEL
LIN {X 0,Y 291.543,Z 488.17,A -85,B 0,C 180,E1 -16724.623,E2 -16724.623} C_VEL
LIN {X 0,Y 291.524,Z 488.162,A -85,B 0,C 180,E1 -16728.88,E2 -16728.88} C_VEL
LIN {X 0,Y 291.695,Z 488.145,A -85,B 0,C 180,E1 -16731.688,E2 -16731.688} C_VEL
LIN {X 0,Y 291.616,Z 488.162,A -85,B 0,C 180,E1 -16734.468,E2 -16734.468} C_VEL
LIN {X 0,Y 291.876,Z 488.118,A -85,B 0,C 180,E1 -16738.62,E2 -16738.62} C_VEL
LIN {X 0,Y 291.878,Z 488.122,A -85,B 0,C 180,E1 -16741.379,E2 -16741.379} C_VEL
LIN {X 0,Y 291.732,Z 488.138,A -85,B 0,C 180,E1 -16746.918,E2 -16746.918} C_VEL
LIN {X 0,Y 291.616,Z 488.148,A -85,B 0,C 180,E1 -16749.712,E2 -16749.712} C_VEL
LIN {X 0,Y 291.508,Z 488.171,A -85,B 0,C 180,E1 -16753.95,E2 -16753.95} C_VEL
LIN {X 0,Y 291.473,Z 488.174,A -85,B 0,C 180,E1 -16756.818,E2 -16756.818} C_VEL
LIN {X 0,Y 291.437,Z 488.17,A -85,B 0,C 180,E1 -16759.875,E2 -16759.875} C_VEL
LIN {X 0,Y 291.387,Z 488.187,A -85,B 0,C 180,E1 -16764.206,E2 -16764.206} C_VEL
LIN {X 0,Y 291.412,Z 488.178,A -85,B 0,C 180,E1 -16767.272,E2 -16767.272} C_VEL
LIN {X 0,Y 291.324,Z 488.189,A -85,B 0,C 180,E1 -16770.438,E2 -16770.438} C_VEL
LIN {X 0,Y 291.332,Z 488.193,A -85,B 0,C 180,E1 -16773.699,E2 -16773.699} C_VEL
LIN {X 0,Y 291.36,Z 488.184,A -85,B 0,C 180,E1 -16777.254,E2 -16777.254} C_VEL
LIN {X 0,Y 291.321,Z 488.197,A -85,B 0,C 180,E1 -16780.644,E2 -16780.644} C_VEL
LIN {X 0,Y 291.331,Z 488.191,A -85,B 0,C 180,E1 -16784.393,E2 -16784.393} C_VEL
LIN {X 0,Y 291.378,Z 488.189,A -85,B 0,C 180,E1 -16788.392,E2 -16788.392} C_VEL
LIN {X 0,Y 291.379,Z 488.18,A -85,B 0,C 180,E1 -16791.166,E2 -16791.166} C_VEL
LIN {X 0,Y 291.377,Z 488.173,A -85,B 0,C 180,E1 -16794.631,E2 -16794.631} C_VEL
LIN {X 0,Y 291.363,Z 488.189,A -85,B 0,C 180,E1 -16797.953,E2 -16797.953} C_VEL
LIN {X 0,Y 291.374,Z 488.18,A -85,B 0,C 180,E1 -16801.16,E2 -16801.16} C_VEL
LIN {X 0,Y 291.409,Z 488.182,A -85,B 0,C 180,E1 -16804.274,E2 -16804.274} C_VEL
LIN {X 0,Y 291.375,Z 488.184,A -85,B 0,C 180,E1 -16807.302,E2 -16807.302} C_VEL
LIN {X 0,Y 291.452,Z 488.18,A -85,B 0,C 180,E1 -16810.272,E2 -16810.272} C_VEL
LIN {X 0,Y 291.55,Z 488.168,A -85,B 0,C 180,E1 -16814.626,E2 -16814.626} C_VEL
LIN {X 0,Y 291.563,Z 488.307,A -85,B 0,C 180,E1 -16818.928,E2 -16818.928} C_VEL
LIN {X 0,Y 291.746,Z 489.1,A -85,B 0,C 180,E1 -16819.154,E2 -16819.154} C_VEL
LIN {X 0,Y 299.127,Z 506.924,A -85,B 0,C 180,E1 -16820.193,E2 -16820.193} C_VEL
LIN {X 0,Y 301.507,Z 513.566,A -85,B 0,C 180,E1 -16820.528,E2 -16820.528} C_VEL
LIN {X 0,Y 300.62,Z 559.993,A -85,B 0,C 180,E1 -16821.633,E2 -16821.633} C_VEL
LIN {X 0,Y 300.483,Z 575.61,A -85,B 0,C 180,E1 -16822.104,E2 -16822.104} C_VEL
LIN {X 0,Y 300.205,Z 588.462,A -85,B 0,C 180,E1 -16822.774,E2 -16822.774} C_VEL
LIN {X 0,Y 299.64,Z 599.85,A -85,B 0,C 180,E1 -16823.606,E2 -16823.606} C_VEL
LIN {X 0,Y 298.795,Z 611.957,A -85,B 0,C 180,E1 -16824.773,E2 -16824.773} C_VEL
LIN {X 0,Y 297.826,Z 622.811,A -85,B 0,C 180,E1 -16826.112,E2 -16826.112} C_VEL
LIN {X 0,Y 296.752,Z 632.626,A -85,B 0,C 180,E1 -16827.627,E2 -16827.627} C_VEL
LIN {X 0,Y 295.635,Z 641.826,A -85,B 0,C 180,E1 -16829.378,E2 -16829.378} C_VEL
LIN {X 0,Y 294.568,Z 650.289,A -85,B 0,C 180,E1 -16831.369,E2 -16831.369} C_VEL
LIN {X 0,Y 293.63,Z 657.286,A -85,B 0,C 180,E1 -16833.433,E2 -16833.433} C_VEL
LIN {X 0,Y 292.92,Z 662.883,A -85,B 0,C 180,E1 -16835.509,E2 -16835.509} C_VEL
LIN {X 0,Y 292.382,Z 667.304,A -85,B 0,C 180,E1 -16837.599,E2 -16837.599} C_VEL
LIN {X 0,Y 291.938,Z 670.677,A -85,B 0,C 180,E1 -16839.704,E2 -16839.704} C_VEL
LIN {X 0,Y 291.813,Z 672.357,A -85,B 0,C 180,E1 -16841.111,E2 -16841.111} C_VEL
LIN {X 0,Y 291.739,Z 673.643,A -85,B 0,C 180,E1 -16842.524,E2 -16842.524} C_VEL
LIN {X 0,Y 291.765,Z 674.485,A -85,B 0,C 180,E1 -16843.941,E2 -16843.941} C_VEL
LIN {X 0,Y 291.976,Z 674.962,A -85,B 0,C 180,E1 -16845.675,E2 -16845.675} C_VEL
LIN {X 0,Y 292.458,Z 674.597,A -85,B 0,C 180,E1 -16848.206,E2 -16848.206} C_VEL
LIN {X 0,Y 293.265,Z 672.784,A -85,B 0,C 180,E1 -16850.834,E2 -16850.834} C_VEL
LIN {X 0,Y 294.355,Z 669.88,A -85,B 0,C 180,E1 -16853.203,E2 -16853.203} C_VEL
LIN {X 0,Y 295.623,Z 666.008,A -85,B 0,C 180,E1 -16855.393,E2 -16855.393} C_VEL
LIN {X 0,Y 297.059,Z 661.129,A -85,B 0,C 180,E1 -16857.476,E2 -16857.476} C_VEL
LIN {X 0,Y 298.833,Z 654.724,A -85,B 0,C 180,E1 -16859.598,E2 -16859.598} C_VEL
LIN {X 0,Y 300.785,Z 646.566,A -85,B 0,C 180,E1 -16861.719,E2 -16861.719} C_VEL
LIN {X 0,Y 302.851,Z 637.385,A -85,B 0,C 180,E1 -16863.606,E2 -16863.606} C_VEL
LIN {X 0,Y 304.644,Z 627.527,A -85,B 0,C 180,E1 -16865.224,E2 -16865.224} C_VEL
LIN {X 0,Y 306.402,Z 616.85,A -85,B 0,C 180,E1 -16866.613,E2 -16866.613} C_VEL
LIN {X 0,Y 307.682,Z 606.783,A -85,B 0,C 180,E1 -16867.665,E2 -16867.665} C_VEL
LIN {X 0,Y 308.763,Z 594.548,A -85,B 0,C 180,E1 -16868.671,E2 -16868.671} C_VEL
LIN {X 0,Y 309.509,Z 581.326,A -85,B 0,C 180,E1 -16869.439,E2 -16869.439} C_VEL
LIN {X 0,Y 309.75,Z 568.993,A -85,B 0,C 180,E1 -16869.913,E2 -16869.913} C_VEL
LIN {X 0,Y 310.67,Z 527.847,A -85,B 0,C 180,E1 -16870.924,E2 -16870.924} C_VEL
LIN {X 0,Y 310.664,Z 523.884,A -85,B 0,C 180,E1 -16871.033,E2 -16871.033} C_VEL
LIN {X 0,Y 302.683,Z 508.392,A -85,B 0,C 180,E1 -16872.445,E2 -16872.445} C_VEL
LIN {X 0,Y 294.858,Z 495.041,A -85,B 0,C 180,E1 -16873.877,E2 -16873.877} C_VEL
LIN {X 0,Y 293.342,Z 492.582,A -85,B 0,C 180,E1 -16874.173,E2 -16874.173} C_VEL
LIN {X 0,Y 292.344,Z 491.684,A -85,B 0,C 180,E1 -16874.473,E2 -16874.473} C_VEL
LIN {X 0,Y 292.23,Z 492.022,A -85,B 0,C 180,E1 -16874.811,E2 -16874.811} C_VEL
LIN {X 0,Y 295.511,Z 505.733,A -85,B 0,C 180,E1 -16877.994,E2 -16877.994} C_VEL
LIN {X 0,Y 297.642,Z 516.602,A -85,B 0,C 180,E1 -16880.393,E2 -16880.393} C_VEL
LIN {X 0,Y 296.98,Z 526.623,A -85,B 0,C 180,E1 -16882.369,E2 -16882.369} C_VEL
LIN {X 0,Y 300.466,Z 553.568,A -85,B 0,C 180,E1 -16883.491,E2 -16883.491} C_VEL
LIN {X 0,Y 300.447,Z 554.417,A -85,B 0,C 180,E1 -16883.518,E2 -16883.518} C_VEL
LIN {X 0,Y 299.692,Z 560.21,A -85,B 0,C 180,E1 -16883.674,E2 -16883.674} C_VEL
LIN {X 0,Y 293.32,Z 578.951,A -85,B 0,C 180,E1 -16883.987,E2 -16883.987} C_VEL
LIN {X 0,Y 292.407,Z 584.748,A -85,B 0,C 180,E1 -16884.143,E2 -16884.143} C_VEL
LIN {X 0,Y 290.476,Z 639.523,A -85,B 0,C 180,E1 -16885.965,E2 -16885.965} C_VEL
LIN {X 0,Y 289.78,Z 653.337,A -85,B 0,C 180,E1 -16886.721,E2 -16886.721} C_VEL
LIN {X 0,Y 288.938,Z 665.532,A -85,B 0,C 180,E1 -16887.649,E2 -16887.649} C_VEL
LIN {X 0,Y 288.07,Z 676.915,A -85,B 0,C 180,E1 -16888.773,E2 -16888.773} C_VEL
LIN {X 0,Y 286.958,Z 688.843,A -85,B 0,C 180,E1 -16890.268,E2 -16890.268} C_VEL
LIN {X 0,Y 285.891,Z 699.604,A -85,B 0,C 180,E1 -16891.957,E2 -16891.957} C_VEL
LIN {X 0,Y 284.806,Z 710.152,A -85,B 0,C 180,E1 -16894.024,E2 -16894.024} C_VEL
LIN {X 0,Y 284.077,Z 717.801,A -85,B 0,C 180,E1 -16895.885,E2 -16895.885} C_VEL
LIN {X 0,Y 283.362,Z 725.301,A -85,B 0,C 180,E1 -16898.16,E2 -16898.16} C_VEL
LIN {X 0,Y 282.905,Z 730.896,A -85,B 0,C 180,E1 -16900.299,E2 -16900.299} C_VEL
LIN {X 0,Y 282.584,Z 735.586,A -85,B 0,C 180,E1 -16902.636,E2 -16902.636} C_VEL
LIN {X 0,Y 282.452,Z 737.839,A -85,B 0,C 180,E1 -16904.116,E2 -16904.116} C_VEL
LIN {X 0,Y 282.453,Z 740.052,A -85,B 0,C 180,E1 -16906.032,E2 -16906.032} C_VEL
LIN {X 0,Y 282.511,Z 741.741,A -85,B 0,C 180,E1 -16908.521,E2 -16908.521} C_VEL
LIN {X 0,Y 282.697,Z 742.145,A -85,B 0,C 180,E1 -16909.979,E2 -16909.979} C_VEL
LIN {X 0,Y 282.974,Z 742.059,A -85,B 0,C 180,E1 -16911.431,E2 -16911.431} C_VEL
LIN {X 0,Y 283.356,Z 741.548,A -85,B 0,C 180,E1 -16912.877,E2 -16912.877} C_VEL
LIN {X 0,Y 283.819,Z 740.632,A -85,B 0,C 180,E1 -16914.316,E2 -16914.316} C_VEL
LIN {X 0,Y 284.296,Z 739.257,A -85,B 0,C 180,E1 -16915.747,E2 -16915.747} C_VEL
LIN {X 0,Y 285.297,Z 736.362,A -85,B 0,C 180,E1 -16917.883,E2 -16917.883} C_VEL
LIN {X 0,Y 286.671,Z 732.358,A -85,B 0,C 180,E1 -16920.001,E2 -16920.001} C_VEL
LIN {X 0,Y 288.355,Z 727.1,A -85,B 0,C 180,E1 -16922.123,E2 -16922.123} C_VEL
LIN {X 0,Y 290.357,Z 720.682,A -85,B 0,C 180,E1 -16924.165,E2 -16924.165} C_VEL
LIN {X 0,Y 292.638,Z 712.601,A -85,B 0,C 180,E1 -16926.205,E2 -16926.205} C_VEL
LIN {X 0,Y 295.226,Z 702.504,A -85,B 0,C 180,E1 -16928.212,E2 -16928.212} C_VEL
LIN {X 0,Y 297.705,Z 692.021,A -85,B 0,C 180,E1 -16929.855,E2 -16929.855} C_VEL
LIN {X 0,Y 299.756,Z 681.837,A -85,B 0,C 180,E1 -16931.153,E2 -16931.153} C_VEL
LIN {X 0,Y 301.712,Z 670.658,A -85,B 0,C 180,E1 -16932.29,E2 -16932.29} C_VEL
LIN {X 0,Y 303.504,Z 657.617,A -85,B 0,C 180,E1 -16933.305,E2 -16933.305} C_VEL
LIN {X 0,Y 304.87,Z 644.551,A -85,B 0,C 180,E1 -16934.044,E2 -16934.044} C_VEL
LIN {X 0,Y 311.109,Z 570.683,A -85,B 0,C 180,E1 -16936.699,E2 -16936.699} C_VEL
LIN {X 0,Y 311.708,Z 562.331,A -85,B 0,C 180,E1 -16937.022,E2 -16937.022} C_VEL
LIN {X 0,Y 309.436,Z 548.534,A -85,B 0,C 180,E1 -16938.274,E2 -16938.274} C_VEL
LIN {X 0,Y 308.588,Z 545.195,A -85,B 0,C 180,E1 -16938.653,E2 -16938.653} C_VEL
LIN {X 0,Y 304.599,Z 536.799,A -85,B 0,C 180,E1 -16940.117,E2 -16940.117} C_VEL
LIN {X 0,Y 303.012,Z 533.525,A -85,B 0,C 180,E1 -16940.797,E2 -16940.797} C_VEL
LIN {X 0,Y 301.784,Z 527.975,A -85,B 0,C 180,E1 -16942.82,E2 -16942.82} C_VEL
LIN {X 0,Y 299.989,Z 521.284,A -85,B 0,C 180,E1 -16945.685,E2 -16945.685} C_VEL
LIN {X 0,Y 298.504,Z 516.673,A -85,B 0,C 180,E1 -16948.092,E2 -16948.092} C_VEL
LIN {X 0,Y 297.081,Z 512.796,A -85,B 0,C 180,E1 -16950.605,E2 -16950.605} C_VEL
LIN {X 0,Y 295.324,Z 508.457,A -85,B 0,C 180,E1 -16954.831,E2 -16954.831} C_VEL
LIN {X 0,Y 294.885,Z 507.541,A -85,B 0,C 180,E1 -16956.572,E2 -16956.572} C_VEL
LIN {X 0,Y 294.802,Z 507.033,A -85,B 0,C 180,E1 -16960.067,E2 -16960.067} C_VEL
LIN {X 0,Y 295.823,Z 508.247,A -85,B 0,C 180,E1 -16963.549,E2 -16963.549} C_VEL
LIN {X 0,Y 296.858,Z 509.394,A -85,B 0,C 180,E1 -16965.255,E2 -16965.255} C_VEL
LIN {X 0,Y 298.53,Z 512.231,A -85,B 0,C 180,E1 -16967.578,E2 -16967.578} C_VEL
LIN {X 0,Y 299.361,Z 514.898,A -85,B 0,C 180,E1 -16968.9,E2 -16968.9} C_VEL
LIN {X 0,Y 300.5,Z 521.531,A -85,B 0,C 180,E1 -16971.099,E2 -16971.099} C_VEL
LIN {X 0,Y 302.305,Z 530.691,A -85,B 0,C 180,E1 -16973.559,E2 -16973.559} C_VEL
LIN {X 0,Y 304.072,Z 538.399,A -85,B 0,C 180,E1 -16975.315,E2 -16975.315} C_VEL
LIN {X 0,Y 303.994,Z 547.13,A -85,B 0,C 180,E1 -16976.527,E2 -16976.527} C_VEL
LIN {X 0,Y 305.934,Z 563.05,A -85,B 0,C 180,E1 -16977.968,E2 -16977.968} C_VEL
LIN {X 0,Y 307.528,Z 581.368,A -85,B 0,C 180,E1 -16979.349,E2 -16979.349} C_VEL
LIN {X 0,Y 308.06,Z 596.071,A -85,B 0,C 180,E1 -16980.239,E2 -16980.239} C_VEL
LIN {X 0,Y 308.001,Z 608.763,A -85,B 0,C 180,E1 -16980.886,E2 -16980.886} C_VEL
LIN {X 0,Y 302.956,Z 669.863,A -85,B 0,C 180,E1 -16983.102,E2 -16983.102} C_VEL
LIN {X 0,Y 301.224,Z 683.959,A -85,B 0,C 180,E1 -16983.87,E2 -16983.87} C_VEL
LIN {X 0,Y 298.773,Z 698.182,A -85,B 0,C 180,E1 -16984.948,E2 -16984.948} C_VEL
LIN {X 0,Y 296.385,Z 710.538,A -85,B 0,C 180,E1 -16986.225,E2 -16986.225} C_VEL
LIN {X 0,Y 293.661,Z 722.922,A -85,B 0,C 180,E1 -16987.854,E2 -16987.854} C_VEL
LIN {X 0,Y 291.227,Z 732.911,A -85,B 0,C 180,E1 -16989.515,E2 -16989.515} C_VEL
LIN {X 0,Y 288.773,Z 742.71,A -85,B 0,C 180,E1 -16991.553,E2 -16991.553} C_VEL
LIN {X 0,Y 287.011,Z 749.41,A -85,B 0,C 180,E1 -16993.276,E2 -16993.276} C_VEL
LIN {X 0,Y 285.755,Z 755.067,A -85,B 0,C 180,E1 -16995.032,E2 -16995.032} C_VEL
LIN {X 0,Y 284.272,Z 760.659,A -85,B 0,C 180,E1 -16997.141,E2 -16997.141} C_VEL
LIN {X 0,Y 283.422,Z 765.029,A -85,B 0,C 180,E1 -16999.28,E2 -16999.28} C_VEL
LIN {X 0,Y 282.813,Z 768.319,A -85,B 0,C 180,E1 -17001.423,E2 -17001.423} C_VEL
LIN {X 0,Y 282.597,Z 769.941,A -85,B 0,C 180,E1 -17002.855,E2 -17002.855} C_VEL
LIN {X 0,Y 282.526,Z 771.139,A -85,B 0,C 180,E1 -17004.287,E2 -17004.287} C_VEL
LIN {X 0,Y 282.543,Z 771.923,A -85,B 0,C 180,E1 -17005.718,E2 -17005.718} C_VEL
LIN {X 0,Y 282.582,Z 772.253,A -85,B 0,C 180,E1 -17007.146,E2 -17007.146} C_VEL
LIN {X 0,Y 282.716,Z 772.127,A -85,B 0,C 180,E1 -17008.573,E2 -17008.573} C_VEL
LIN {X 0,Y 282.964,Z 771.586,A -85,B 0,C 180,E1 -17009.998,E2 -17009.998} C_VEL
LIN {X 0,Y 282.883,Z 770.579,A -85,B 0,C 180,E1 -17011.421,E2 -17011.421} C_VEL
LIN {X 0,Y 282.7,Z 769.047,A -85,B 0,C 180,E1 -17012.848,E2 -17012.848} C_VEL
LIN {X 0,Y 282.775,Z 765.872,A -85,B 0,C 180,E1 -17014.988,E2 -17014.988} C_VEL
LIN {X 0,Y 282.765,Z 761.47,A -85,B 0,C 180,E1 -17017.136,E2 -17017.136} C_VEL
LIN {X 0,Y 282.993,Z 755.749,A -85,B 0,C 180,E1 -17019.287,E2 -17019.287} C_VEL
LIN {X 0,Y 283.397,Z 748.466,A -85,B 0,C 180,E1 -17021.44,E2 -17021.44} C_VEL
LIN {X 0,Y 284.037,Z 740.974,A -85,B 0,C 180,E1 -17023.228,E2 -17023.228} C_VEL
LIN {X 0,Y 285.002,Z 730.872,A -85,B 0,C 180,E1 -17025.187,E2 -17025.187} C_VEL
LIN {X 0,Y 286.013,Z 720.257,A -85,B 0,C 180,E1 -17026.825,E2 -17026.825} C_VEL
LIN {X 0,Y 287.145,Z 709.291,A -85,B 0,C 180,E1 -17028.181,E2 -17028.181} C_VEL
LIN {X 0,Y 288.344,Z 695.435,A -85,B 0,C 180,E1 -17029.578,E2 -17029.578} C_VEL
LIN {X 0,Y 289.828,Z 684.252,A -85,B 0,C 180,E1 -17030.769,E2 -17030.769} C_VEL
LIN {X 0,Y 290.968,Z 672.986,A -85,B 0,C 180,E1 -17031.704,E2 -17031.704} C_VEL
LIN {X 0,Y 291.915,Z 660.523,A -85,B 0,C 180,E1 -17032.467,E2 -17032.467} C_VEL
LIN {X 0,Y 292.536,Z 647.829,A -85,B 0,C 180,E1 -17032.971,E2 -17032.971} C_VEL
LIN {X 0,Y 293.385,Z 602.216,A -85,B 0,C 180,E1 -17034.1,E2 -17034.1} C_VEL
LIN {X 0,Y 287.795,Z 539.429,A -85,B 0,C 180,E1 -17036.146,E2 -17036.146} C_VEL
LIN {X 0,Y 289.189,Z 527.741,A -85,B 0,C 180,E1 -17038.681,E2 -17038.681} C_VEL
LIN {X 0,Y 290.469,Z 517.67,A -85,B 0,C 180,E1 -17040.929,E2 -17040.929} C_VEL
LIN {X 0,Y 287.94,Z 504.789,A -85,B 0,C 180,E1 -17044.148,E2 -17044.148} C_VEL
LIN {X 0,Y 285.131,Z 492.479,A -85,B 0,C 180,E1 -17047.405,E2 -17047.405} C_VEL
LIN {X 0,Y 284.291,Z 489.165,A -85,B 0,C 180,E1 -17048.394,E2 -17048.394} C_VEL
LIN {X 0,Y 284.23,Z 489.082,A -85,B 0,C 180,E1 -17052.115,E2 -17052.115} C_VEL
LIN {X 0,Y 284.247,Z 489.076,A -85,B 0,C 180,E1 -17056.187,E2 -17056.187} C_VEL
LIN {X 0,Y 284.297,Z 489.069,A -85,B 0,C 180,E1 -17060.022,E2 -17060.022} C_VEL
LIN {X 0,Y 284.311,Z 489.069,A -85,B 0,C 180,E1 -17063.61,E2 -17063.61} C_VEL
LIN {X 0,Y 284.298,Z 489.069,A -85,B 0,C 180,E1 -17067.188,E2 -17067.188} C_VEL
LIN {X 0,Y 284.348,Z 489.061,A -85,B 0,C 180,E1 -17070.374,E2 -17070.374} C_VEL
LIN {X 0,Y 284.364,Z 489.056,A -85,B 0,C 180,E1 -17073.585,E2 -17073.585} C_VEL
LIN {X 0,Y 284.355,Z 489.064,A -85,B 0,C 180,E1 -17076.705,E2 -17076.705} C_VEL
LIN {X 0,Y 284.391,Z 489.053,A -85,B 0,C 180,E1 -17081.26,E2 -17081.26} C_VEL
LIN {X 0,Y 284.48,Z 489.051,A -85,B 0,C 180,E1 -17084.458,E2 -17084.458} C_VEL
LIN {X 0,Y 284.476,Z 489.039,A -85,B 0,C 180,E1 -17088.6,E2 -17088.6} C_VEL
LIN {X 0,Y 284.646,Z 489.023,A -85,B 0,C 180,E1 -17091.48,E2 -17091.48} C_VEL
LIN {X 0,Y 284.587,Z 489.036,A -85,B 0,C 180,E1 -17094.33,E2 -17094.33} C_VEL
LIN {X 0,Y 284.842,Z 488.992,A -85,B 0,C 180,E1 -17098.586,E2 -17098.586} C_VEL
LIN {X 0,Y 284.843,Z 488.998,A -85,B 0,C 180,E1 -17101.413,E2 -17101.413} C_VEL
LIN {X 0,Y 284.684,Z 489.014,A -85,B 0,C 180,E1 -17107.09,E2 -17107.09} C_VEL
LIN {X 0,Y 284.553,Z 489.027,A -85,B 0,C 180,E1 -17109.955,E2 -17109.955} C_VEL
LIN {X 0,Y 284.468,Z 489.05,A -85,B 0,C 180,E1 -17114.303,E2 -17114.303} C_VEL
LIN {X 0,Y 284.412,Z 489.05,A -85,B 0,C 180,E1 -17117.249,E2 -17117.249} C_VEL
LIN {X 0,Y 284.365,Z 489.051,A -85,B 0,C 180,E1 -17120.243,E2 -17120.243} C_VEL
LIN {X 0,Y 284.356,Z 489.061,A -85,B 0,C 180,E1 -17123.876,E2 -17123.876} C_VEL
LIN {X 0,Y 284.386,Z 489.053,A -85,B 0,C 180,E1 -17127.175,E2 -17127.175} C_VEL
LIN {X 0,Y 284.283,Z 489.071,A -85,B 0,C 180,E1 -17131.275,E2 -17131.275} C_VEL
LIN {X 0,Y 284.328,Z 489.063,A -85,B 0,C 180,E1 -17135.349,E2 -17135.349} C_VEL
LIN {X 0,Y 284.296,Z 489.063,A -85,B 0,C 180,E1 -17138.171,E2 -17138.171} C_VEL
LIN {X 0,Y 284.272,Z 489.073,A -85,B 0,C 180,E1 -17142.129,E2 -17142.129} C_VEL
LIN {X 0,Y 284.307,Z 489.066,A -85,B 0,C 180,E1 -17146.203,E2 -17146.203} C_VEL
LIN {X 0,Y 284.341,Z 489.061,A -85,B 0,C 180,E1 -17150.015,E2 -17150.015} C_VEL
LIN {X 0,Y 284.347,Z 489.043,A -85,B 0,C 180,E1 -17153.62,E2 -17153.62} C_VEL
LIN {X 0,Y 284.299,Z 489.072,A -85,B 0,C 180,E1 -17157.191,E2 -17157.191} C_VEL
LIN {X 0,Y 284.35,Z 489.061,A -85,B 0,C 180,E1 -17160.378,E2 -17160.378} C_VEL
LIN {X 0,Y 284.371,Z 489.057,A -85,B 0,C 180,E1 -17163.589,E2 -17163.589} C_VEL
LIN {X 0,Y 284.36,Z 489.064,A -85,B 0,C 180,E1 -17166.709,E2 -17166.709} C_VEL
LIN {X 0,Y 284.398,Z 489.061,A -85,B 0,C 180,E1 -17171.264,E2 -17171.264} C_VEL
LIN {X 0,Y 284.487,Z 489.047,A -85,B 0,C 180,E1 -17174.461,E2 -17174.461} C_VEL
LIN {X 0,Y 284.504,Z 489.244,A -85,B 0,C 180,E1 -17178.424,E2 -17178.424} C_VEL
LIN {X 0,Y 284.77,Z 490.382,A -85,B 0,C 180,E1 -17178.662,E2 -17178.662} C_VEL
LIN {X 0,Y 292.243,Z 508.022,A -85,B 0,C 180,E1 -17179.72,E2 -17179.72} C_VEL
LIN {X 0,Y 294.822,Z 514.953,A -85,B 0,C 180,E1 -17180.089,E2 -17180.089} C_VEL
LIN {X 0,Y 293.925,Z 559.625,A -85,B 0,C 180,E1 -17181.176,E2 -17181.176} C_VEL
LIN {X 0,Y 293.767,Z 576.357,A -85,B 0,C 180,E1 -17181.683,E2 -17181.683} C_VEL
LIN {X 0,Y 293.477,Z 589.015,A -85,B 0,C 180,E1 -17182.347,E2 -17182.347} C_VEL
LIN {X 0,Y 292.867,Z 601.453,A -85,B 0,C 180,E1 -17183.284,E2 -17183.284} C_VEL
LIN {X 0,Y 291.98,Z 613.434,A -85,B 0,C 180,E1 -17184.477,E2 -17184.477} C_VEL
LIN {X 0,Y 290.914,Z 624.185,A -85,B 0,C 180,E1 -17185.846,E2 -17185.846} C_VEL
LIN {X 0,Y 289.947,Z 632.957,A -85,B 0,C 180,E1 -17187.224,E2 -17187.224} C_VEL
LIN {X 0,Y 288.737,Z 642.685,A -85,B 0,C 180,E1 -17189.105,E2 -17189.105} C_VEL
LIN {X 0,Y 287.68,Z 650.685,A -85,B 0,C 180,E1 -17191.017,E2 -17191.017} C_VEL
LIN {X 0,Y 286.709,Z 657.924,A -85,B 0,C 180,E1 -17193.164,E2 -17193.164} C_VEL
LIN {X 0,Y 285.83,Z 664.41,A -85,B 0,C 180,E1 -17195.647,E2 -17195.647} C_VEL
LIN {X 0,Y 285.317,Z 668.707,A -85,B 0,C 180,E1 -17197.789,E2 -17197.789} C_VEL
LIN {X 0,Y 284.881,Z 671.969,A -85,B 0,C 180,E1 -17199.947,E2 -17199.947} C_VEL
LIN {X 0,Y 284.764,Z 673.597,A -85,B 0,C 180,E1 -17201.39,E2 -17201.39} C_VEL
LIN {X 0,Y 284.708,Z 674.798,A -85,B 0,C 180,E1 -17202.839,E2 -17202.839} C_VEL
LIN {X 0,Y 284.957,Z 675.941,A -85,B 0,C 180,E1 -17205.744,E2 -17205.744} C_VEL
LIN {X 0,Y 285.198,Z 675.932,A -85,B 0,C 180,E1 -17207.202,E2 -17207.202} C_VEL
LIN {X 0,Y 285.535,Z 675.473,A -85,B 0,C 180,E1 -17208.664,E2 -17208.664} C_VEL
LIN {X 0,Y 286.389,Z 673.72,A -85,B 0,C 180,E1 -17211.17,E2 -17211.17} C_VEL
LIN {X 0,Y 287.656,Z 670.529,A -85,B 0,C 180,E1 -17213.776,E2 -17213.776} C_VEL
LIN {X 0,Y 288.967,Z 666.639,A -85,B 0,C 180,E1 -17215.965,E2 -17215.965} C_VEL
LIN {X 0,Y 290.849,Z 660.483,A -85,B 0,C 180,E1 -17218.507,E2 -17218.507} C_VEL
LIN {X 0,Y 292.804,Z 653.644,A -85,B 0,C 180,E1 -17220.67,E2 -17220.67} C_VEL
LIN {X 0,Y 294.554,Z 646.558,A -85,B 0,C 180,E1 -17222.472,E2 -17222.472} C_VEL
LIN {X 0,Y 296.634,Z 637.464,A -85,B 0,C 180,E1 -17224.325,E2 -17224.325} C_VEL
LIN {X 0,Y 298.593,Z 626.912,A -85,B 0,C 180,E1 -17226.048,E2 -17226.048} C_VEL
LIN {X 0,Y 300.493,Z 615.855,A -85,B 0,C 180,E1 -17227.454,E2 -17227.454} C_VEL
LIN {X 0,Y 301.886,Z 604.173,A -85,B 0,C 180,E1 -17228.626,E2 -17228.626} C_VEL
LIN {X 0,Y 302.913,Z 592.314,A -85,B 0,C 180,E1 -17229.532,E2 -17229.532} C_VEL
LIN {X 0,Y 303.515,Z 579.562,A -85,B 0,C 180,E1 -17230.239,E2 -17230.239} C_VEL
LIN {X 0,Y 303.758,Z 566.486,A -85,B 0,C 180,E1 -17230.682,E2 -17230.682} C_VEL
LIN {X 0,Y 304.683,Z 526.22,A -85,B 0,C 180,E1 -17231.691,E2 -17231.691} C_VEL
LIN {X 0,Y 296.501,Z 510.391,A -85,B 0,C 180,E1 -17233.199,E2 -17233.199} C_VEL
LIN {X 0,Y 289.832,Z 499.097,A -85,B 0,C 180,E1 -17234.471,E2 -17234.471} C_VEL
LIN {X 0,Y 287.307,Z 498.098,A -85,B 0,C 180,E1 -17234.886,E2 -17234.886} C_VEL
LIN {X 0,Y 286.414,Z 497.303,A -85,B 0,C 180,E1 -17235.196,E2 -17235.196} C_VEL
LIN {X 0,Y 286.337,Z 497.564,A -85,B 0,C 180,E1 -17235.487,E2 -17235.487} C_VEL
LIN {X 0,Y 289.124,Z 509.816,A -85,B 0,C 180,E1 -17238.374,E2 -17238.374} C_VEL
LIN {X 0,Y 290.679,Z 517.423,A -85,B 0,C 180,E1 -17240.077,E2 -17240.077} C_VEL
LIN {X 0,Y 290.136,Z 527.121,A -85,B 0,C 180,E1 -17242,E2 -17242} C_VEL
LIN {X 0,Y 293.601,Z 554.046,A -85,B 0,C 180,E1 -17243.148,E2 -17243.148} C_VEL
LIN {X 0,Y 292.407,Z 584.748,A -85,B 0,C 180,E1 -17244.143,E2 -17244.143} C_VEL
LIN {X 0,Y 291.517,Z 590.541,A -85,B 0,C 180,E1 -17244.301,E2 -17244.301} C_VEL
LIN {X 0,Y 285.24,Z 609.292,A -85,B 0,C 180,E1 -17244.648,E2 -17244.648} C_VEL
LIN {X 0,Y 284.413,Z 615.085,A -85,B 0,C 180,E1 -17244.813,E2 -17244.813} C_VEL
LIN {X 0,Y 283.466,Z 640.612,A -85,B 0,C 180,E1 -17245.719,E2 -17245.719} C_VEL
LIN {X 0,Y 282.768,Z 654.689,A -85,B 0,C 180,E1 -17246.534,E2 -17246.534} C_VEL
LIN {X 0,Y 281.837,Z 667.883,A -85,B 0,C 180,E1 -17247.604,E2 -17247.604} C_VEL
LIN {X 0,Y 280.766,Z 680.194,A -85,B 0,C 180,E1 -17248.918,E2 -17248.918} C_VEL
LIN {X 0,Y 279.691,Z 691.54,A -85,B 0,C 180,E1 -17250.454,E2 -17250.454} C_VEL
LIN {X 0,Y 278.546,Z 702.721,A -85,B 0,C 180,E1 -17252.349,E2 -17252.349} C_VEL
LIN {X 0,Y 277.658,Z 711.164,A -85,B 0,C 180,E1 -17254.112,E2 -17254.112} C_VEL
LIN {X 0,Y 276.915,Z 718.762,A -85,B 0,C 180,E1 -17256.042,E2 -17256.042} C_VEL
LIN {X 0,Y 276.214,Z 726.114,A -85,B 0,C 180,E1 -17258.35,E2 -17258.35} C_VEL
LIN {X 0,Y 275.795,Z 731.885,A -85,B 0,C 180,E1 -17260.654,E2 -17260.654} C_VEL
LIN {X 0,Y 275.45,Z 736.235,A -85,B 0,C 180,E1 -17262.938,E2 -17262.938} C_VEL
LIN {X 0,Y 275.353,Z 740.168,A -85,B 0,C 180,E1 -17265.914,E2 -17265.914} C_VEL
LIN {X 0,Y 275.417,Z 741.923,A -85,B 0,C 180,E1 -17268.221,E2 -17268.221} C_VEL
LIN {X 0,Y 275.576,Z 742.471,A -85,B 0,C 180,E1 -17269.717,E2 -17269.717} C_VEL
LIN {X 0,Y 275.85,Z 742.602,A -85,B 0,C 180,E1 -17271.208,E2 -17271.208} C_VEL
LIN {X 0,Y 276.272,Z 742.248,A -85,B 0,C 180,E1 -17272.813,E2 -17272.813} C_VEL
LIN {X 0,Y 277.186,Z 740.358,A -85,B 0,C 180,E1 -17275.638,E2 -17275.638} C_VEL
LIN {X 0,Y 278.212,Z 737.749,A -85,B 0,C 180,E1 -17277.829,E2 -17277.829} C_VEL
LIN {X 0,Y 279.625,Z 734.103,A -85,B 0,C 180,E1 -17280.001,E2 -17280.001} C_VEL
LIN {X 0,Y 281.326,Z 729.32,A -85,B 0,C 180,E1 -17282.146,E2 -17282.146} C_VEL
LIN {X 0,Y 283.413,Z 723.201,A -85,B 0,C 180,E1 -17284.267,E2 -17284.267} C_VEL
LIN {X 0,Y 285.738,Z 715.591,A -85,B 0,C 180,E1 -17286.355,E2 -17286.355} C_VEL
LIN {X 0,Y 288.475,Z 706.216,A -85,B 0,C 180,E1 -17288.406,E2 -17288.406} C_VEL
LIN {X 0,Y 290.947,Z 696.526,A -85,B 0,C 180,E1 -17290.087,E2 -17290.087} C_VEL
LIN {X 0,Y 293.37,Z 685.858,A -85,B 0,C 180,E1 -17291.574,E2 -17291.574} C_VEL
LIN {X 0,Y 295.851,Z 673.018,A -85,B 0,C 180,E1 -17292.973,E2 -17292.973} C_VEL
LIN {X 0,Y 297.896,Z 659.997,A -85,B 0,C 180,E1 -17294.056,E2 -17294.056} C_VEL
LIN {X 0,Y 299.505,Z 646.485,A -85,B 0,C 180,E1 -17294.874,E2 -17294.874} C_VEL
LIN {X 0,Y 301.166,Z 626.655,A -85,B 0,C 180,E1 -17295.654,E2 -17295.654} C_VEL
LIN {X 0,Y 306.887,Z 564.063,A -85,B 0,C 180,E1 -17297.943,E2 -17297.943} C_VEL
LIN {X 0,Y 304.621,Z 550.007,A -85,B 0,C 180,E1 -17299.287,E2 -17299.287} C_VEL
LIN {X 0,Y 300.931,Z 541.902,A -85,B 0,C 180,E1 -17300.749,E2 -17300.749} C_VEL
LIN {X 0,Y 297.09,Z 534.288,A -85,B 0,C 180,E1 -17302.468,E2 -17302.468} C_VEL
LIN {X 0,Y 295.464,Z 527.531,A -85,B 0,C 180,E1 -17305.351,E2 -17305.351} C_VEL
LIN {X 0,Y 294.111,Z 522.702,A -85,B 0,C 180,E1 -17307.85,E2 -17307.85} C_VEL
LIN {X 0,Y 292.895,Z 518.975,A -85,B 0,C 180,E1 -17310.258,E2 -17310.258} C_VEL
LIN {X 0,Y 291.518,Z 515.302,A -85,B 0,C 180,E1 -17313.676,E2 -17313.676} C_VEL
LIN {X 0,Y 291.147,Z 513.98,A -85,B 0,C 180,E1 -17315.404,E2 -17315.404} C_VEL
LIN {X 0,Y 290.851,Z 513.272,A -85,B 0,C 180,E1 -17317.164,E2 -17317.164} C_VEL
LIN {X 0,Y 291.082,Z 513.148,A -85,B 0,C 180,E1 -17320.686,E2 -17320.686} C_VEL
LIN {X 0,Y 292.478,Z 514.695,A -85,B 0,C 180,E1 -17324.175,E2 -17324.175} C_VEL
LIN {X 0,Y 294.208,Z 517.25,A -85,B 0,C 180,E1 -17326.769,E2 -17326.769} C_VEL
LIN {X 0,Y 295.216,Z 519.645,A -85,B 0,C 180,E1 -17328.194,E2 -17328.194} C_VEL
LIN {X 0,Y 296.068,Z 525.151,A -85,B 0,C 180,E1 -17330.137,E2 -17330.137} C_VEL
LIN {X 0,Y 297.479,Z 533.216,A -85,B 0,C 180,E1 -17332.434,E2 -17332.434} C_VEL
LIN {X 0,Y 299.362,Z 542.095,A -85,B 0,C 180,E1 -17334.582,E2 -17334.582} C_VEL
LIN {X 0,Y 299.262,Z 546.895,A -85,B 0,C 180,E1 -17335.282,E2 -17335.282} C_VEL
LIN {X 0,Y 301.139,Z 563.023,A -85,B 0,C 180,E1 -17336.838,E2 -17336.838} C_VEL
LIN {X 0,Y 302.606,Z 581.3,A -85,B 0,C 180,E1 -17338.296,E2 -17338.296} C_VEL
LIN {X 0,Y 303.081,Z 596.701,A -85,B 0,C 180,E1 -17339.284,E2 -17339.284} C_VEL
LIN {X 0,Y 302.941,Z 609.038,A -85,B 0,C 180,E1 -17339.954,E2 -17339.954} C_VEL
LIN {X 0,Y 297.64,Z 669.482,A -85,B 0,C 180,E1 -17342.2,E2 -17342.2} C_VEL
LIN {X 0,Y 295.766,Z 683.334,A -85,B 0,C 180,E1 -17342.968,E2 -17342.968} C_VEL
LIN {X 0,Y 293.212,Z 697.477,A -85,B 0,C 180,E1 -17344.057,E2 -17344.057} C_VEL
LIN {X 0,Y 290.951,Z 708.539,A -85,B 0,C 180,E1 -17345.182,E2 -17345.182} C_VEL
LIN {X 0,Y 288.048,Z 721.117,A -85,B 0,C 180,E1 -17346.83,E2 -17346.83} C_VEL
LIN {X 0,Y 285.616,Z 730.376,A -85,B 0,C 180,E1 -17348.338,E2 -17348.338} C_VEL
LIN {X 0,Y 282.897,Z 740.492,A -85,B 0,C 180,E1 -17350.402,E2 -17350.402} C_VEL
LIN {X 0,Y 280.543,Z 748.768,A -85,B 0,C 180,E1 -17352.503,E2 -17352.503} C_VEL
LIN {X 0,Y 278.905,Z 755.426,A -85,B 0,C 180,E1 -17354.655,E2 -17354.655} C_VEL
LIN {X 0,Y 277.332,Z 760.798,A -85,B 0,C 180,E1 -17356.814,E2 -17356.814} C_VEL
LIN {X 0,Y 276.418,Z 765.029,A -85,B 0,C 180,E1 -17359.005,E2 -17359.005} C_VEL
LIN {X 0,Y 275.773,Z 768.192,A -85,B 0,C 180,E1 -17361.202,E2 -17361.202} C_VEL
LIN {X 0,Y 275.522,Z 769.732,A -85,B 0,C 180,E1 -17362.67,E2 -17362.67} C_VEL
LIN {X 0,Y 275.451,Z 770.978,A -85,B 0,C 180,E1 -17364.311,E2 -17364.311} C_VEL
LIN {X 0,Y 275.459,Z 771.562,A -85,B 0,C 180,E1 -17365.608,E2 -17365.608} C_VEL
LIN {X 0,Y 275.502,Z 771.795,A -85,B 0,C 180,E1 -17367.073,E2 -17367.073} C_VEL
LIN {X 0,Y 275.627,Z 771.609,A -85,B 0,C 180,E1 -17368.536,E2 -17368.536} C_VEL
LIN {X 0,Y 275.903,Z 771.007,A -85,B 0,C 180,E1 -17369.998,E2 -17369.998} C_VEL
LIN {X 0,Y 275.808,Z 769.877,A -85,B 0,C 180,E1 -17371.458,E2 -17371.458} C_VEL
LIN {X 0,Y 275.632,Z 767.303,A -85,B 0,C 180,E1 -17373.652,E2 -17373.652} C_VEL
LIN {X 0,Y 275.665,Z 763.597,A -85,B 0,C 180,E1 -17375.851,E2 -17375.851} C_VEL
LIN {X 0,Y 275.765,Z 758.624,A -85,B 0,C 180,E1 -17378.055,E2 -17378.055} C_VEL
LIN {X 0,Y 276.076,Z 752.253,A -85,B 0,C 180,E1 -17380.262,E2 -17380.262} C_VEL
LIN {X 0,Y 276.683,Z 744.181,A -85,B 0,C 180,E1 -17382.466,E2 -17382.466} C_VEL
LIN {X 0,Y 277.418,Z 735.862,A -85,B 0,C 180,E1 -17384.298,E2 -17384.298} C_VEL
LIN {X 0,Y 278.367,Z 725.684,A -85,B 0,C 180,E1 -17386.122,E2 -17386.122} C_VEL
LIN {X 0,Y 279.569,Z 714.24,A -85,B 0,C 180,E1 -17387.744,E2 -17387.744} C_VEL
LIN {X 0,Y 280.631,Z 703.128,A -85,B 0,C 180,E1 -17388.997,E2 -17388.997} C_VEL
LIN {X 0,Y 281.224,Z 696.357,A -85,B 0,C 180,E1 -17389.714,E2 -17389.714} C_VEL
LIN {X 0,Y 282.681,Z 685.68,A -85,B 0,C 180,E1 -17390.937,E2 -17390.937} C_VEL
LIN {X 0,Y 284.117,Z 672.812,A -85,B 0,C 180,E1 -17392.064,E2 -17392.064} C_VEL
LIN {X 0,Y 285.139,Z 659.869,A -85,B 0,C 180,E1 -17392.888,E2 -17392.888} C_VEL
LIN {X 0,Y 285.809,Z 646.55,A -85,B 0,C 180,E1 -17393.428,E2 -17393.428} C_VEL
LIN {X 0,Y 286.66,Z 602.81,A -85,B 0,C 180,E1 -17394.533,E2 -17394.533} C_VEL
LIN {X 0,Y 280.974,Z 538.775,A -85,B 0,C 180,E1 -17396.664,E2 -17396.664} C_VEL
LIN {X 0,Y 280.995,Z 537.92,A -85,B 0,C 180,E1 -17396.754,E2 -17396.754} C_VEL
LIN {X 0,Y 283.283,Z 521.175,A -85,B 0,C 180,E1 -17400.567,E2 -17400.567} C_VEL
LIN {X 0,Y 283.359,Z 517.725,A -85,B 0,C 180,E1 -17401.386,E2 -17401.386} C_VEL
LIN {X 0,Y 280.527,Z 503.991,A -85,B 0,C 180,E1 -17404.938,E2 -17404.938} C_VEL
LIN {X 0,Y 277.647,Z 491.739,A -85,B 0,C 180,E1 -17408.307,E2 -17408.307} C_VEL
LIN {X 0,Y 277.245,Z 490.048,A -85,B 0,C 180,E1 -17408.867,E2 -17408.867} C_VEL
LIN {X 0,Y 277.184,Z 489.955,A -85,B 0,C 180,E1 -17413.199,E2 -17413.199} C_VEL
LIN {X 0,Y 277.206,Z 489.953,A -85,B 0,C 180,E1 -17417.323,E2 -17417.323} C_VEL
LIN {X 0,Y 277.244,Z 489.948,A -85,B 0,C 180,E1 -17421.793,E2 -17421.793} C_VEL
LIN {X 0,Y 277.268,Z 489.942,A -85,B 0,C 180,E1 -17424.338,E2 -17424.338} C_VEL
LIN {X 0,Y 277.235,Z 489.95,A -85,B 0,C 180,E1 -17427.835,E2 -17427.835} C_VEL
LIN {X 0,Y 277.259,Z 489.938,A -85,B 0,C 180,E1 -17431.209,E2 -17431.209} C_VEL
LIN {X 0,Y 277.3,Z 489.942,A -85,B 0,C 180,E1 -17434.478,E2 -17434.478} C_VEL
LIN {X 0,Y 277.273,Z 489.944,A -85,B 0,C 180,E1 -17437.653,E2 -17437.653} C_VEL
LIN {X 0,Y 277.333,Z 489.932,A -85,B 0,C 180,E1 -17440.765,E2 -17440.765} C_VEL
LIN {X 0,Y 277.422,Z 489.925,A -85,B 0,C 180,E1 -17445.325,E2 -17445.325} C_VEL
LIN {X 0,Y 277.494,Z 489.907,A -85,B 0,C 180,E1 -17449.788,E2 -17449.788} C_VEL
LIN {X 0,Y 277.639,Z 489.901,A -85,B 0,C 180,E1 -17452.728,E2 -17452.728} C_VEL
LIN {X 0,Y 277.808,Z 489.867,A -85,B 0,C 180,E1 -17458.55,E2 -17458.55} C_VEL
LIN {X 0,Y 277.809,Z 489.874,A -85,B 0,C 180,E1 -17461.449,E2 -17461.449} C_VEL
LIN {X 0,Y 277.639,Z 489.891,A -85,B 0,C 180,E1 -17467.271,E2 -17467.271} C_VEL
LIN {X 0,Y 277.493,Z 489.907,A -85,B 0,C 180,E1 -17470.211,E2 -17470.211} C_VEL
LIN {X 0,Y 277.421,Z 489.93,A -85,B 0,C 180,E1 -17474.674,E2 -17474.674} C_VEL
LIN {X 0,Y 277.331,Z 489.925,A -85,B 0,C 180,E1 -17479.234,E2 -17479.234} C_VEL
LIN {X 0,Y 277.306,Z 489.941,A -85,B 0,C 180,E1 -17484.171,E2 -17484.171} C_VEL
LIN {X 0,Y 277.315,Z 489.932,A -85,B 0,C 180,E1 -17487.507,E2 -17487.507} C_VEL
LIN {X 0,Y 277.259,Z 489.941,A -85,B 0,C 180,E1 -17490.482,E2 -17490.482} C_VEL
LIN {X 0,Y 277.234,Z 489.949,A -85,B 0,C 180,E1 -17493.897,E2 -17493.897} C_VEL
LIN {X 0,Y 277.252,Z 489.939,A -85,B 0,C 180,E1 -17497.471,E2 -17497.471} C_VEL
LIN {X 0,Y 277.204,Z 489.955,A -85,B 0,C 180,E1 -17501.237,E2 -17501.237} C_VEL
LIN {X 0,Y 277.235,Z 489.946,A -85,B 0,C 180,E1 -17505.219,E2 -17505.219} C_VEL
LIN {X 0,Y 277.285,Z 489.941,A -85,B 0,C 180,E1 -17509.496,E2 -17509.496} C_VEL
LIN {X 0,Y 277.282,Z 489.926,A -85,B 0,C 180,E1 -17512.536,E2 -17512.536} C_VEL
LIN {X 0,Y 277.245,Z 489.942,A -85,B 0,C 180,E1 -17516.107,E2 -17516.107} C_VEL
LIN {X 0,Y 277.253,Z 489.946,A -85,B 0,C 180,E1 -17519.541,E2 -17519.541} C_VEL
LIN {X 0,Y 277.351,Z 489.922,A -85,B 0,C 180,E1 -17522.866,E2 -17522.866} C_VEL
LIN {X 0,Y 277.322,Z 489.94,A -85,B 0,C 180,E1 -17526.082,E2 -17526.082} C_VEL
LIN {X 0,Y 277.339,Z 489.941,A -85,B 0,C 180,E1 -17530.769,E2 -17530.769} C_VEL
LIN {X 0,Y 277.43,Z 489.925,A -85,B 0,C 180,E1 -17535.328,E2 -17535.328} C_VEL
LIN {X 0,Y 277.465,Z 490.096,A -85,B 0,C 180,E1 -17537.848,E2 -17537.848} C_VEL
LIN {X 0,Y 277.719,Z 491.2,A -85,B 0,C 180,E1 -17538.103,E2 -17538.103} C_VEL
LIN {X 0,Y 286.069,Z 510.85,A -85,B 0,C 180,E1 -17539.324,E2 -17539.324} C_VEL
LIN {X 0,Y 288.057,Z 516.202,A -85,B 0,C 180,E1 -17539.619,E2 -17539.619} C_VEL
LIN {X 0,Y 287.235,Z 562.789,A -85,B 0,C 180,E1 -17540.789,E2 -17540.789} C_VEL
LIN {X 0,Y 287.087,Z 577.689,A -85,B 0,C 180,E1 -17541.267,E2 -17541.267} C_VEL
LIN {X 0,Y 286.773,Z 589.551,A -85,B 0,C 180,E1 -17541.902,E2 -17541.902} C_VEL
LIN {X 0,Y 286.21,Z 601.118,A -85,B 0,C 180,E1 -17542.773,E2 -17542.773} C_VEL
LIN {X 0,Y 285.27,Z 613.368,A -85,B 0,C 180,E1 -17543.992,E2 -17543.992} C_VEL
LIN {X 0,Y 284.193,Z 624.347,A -85,B 0,C 180,E1 -17545.392,E2 -17545.392} C_VEL
LIN {X 0,Y 283.159,Z 633.264,A -85,B 0,C 180,E1 -17546.801,E2 -17546.801} C_VEL
LIN {X 0,Y 281.842,Z 643.539,A -85,B 0,C 180,E1 -17548.819,E2 -17548.819} C_VEL
LIN {X 0,Y 280.816,Z 651.074,A -85,B 0,C 180,E1 -17550.648,E2 -17550.648} C_VEL
LIN {X 0,Y 279.79,Z 658.54,A -85,B 0,C 180,E1 -17552.882,E2 -17552.882} C_VEL
LIN {X 0,Y 278.985,Z 664.302,A -85,B 0,C 180,E1 -17555.061,E2 -17555.061} C_VEL
LIN {X 0,Y 278.366,Z 668.854,A -85,B 0,C 180,E1 -17557.255,E2 -17557.255} C_VEL
LIN {X 0,Y 277.918,Z 672.41,A -85,B 0,C 180,E1 -17559.521,E2 -17559.521} C_VEL
LIN {X 0,Y 277.708,Z 674.824,A -85,B 0,C 180,E1 -17561.683,E2 -17561.683} C_VEL
LIN {X 0,Y 277.776,Z 676.647,A -85,B 0,C 180,E1 -17564.658,E2 -17564.658} C_VEL
LIN {X 0,Y 277.982,Z 676.974,A -85,B 0,C 180,E1 -17566.149,E2 -17566.149} C_VEL
LIN {X 0,Y 278.276,Z 676.868,A -85,B 0,C 180,E1 -17567.644,E2 -17567.644} C_VEL
LIN {X 0,Y 278.645,Z 676.345,A -85,B 0,C 180,E1 -17569.143,E2 -17569.143} C_VEL
LIN {X 0,Y 279.536,Z 674.649,A -85,B 0,C 180,E1 -17571.529,E2 -17571.529} C_VEL
LIN {X 0,Y 280.961,Z 671.157,A -85,B 0,C 180,E1 -17574.379,E2 -17574.379} C_VEL
LIN {X 0,Y 282.401,Z 667.121,A -85,B 0,C 180,E1 -17576.615,E2 -17576.615} C_VEL
LIN {X 0,Y 284.418,Z 660.808,A -85,B 0,C 180,E1 -17579.213,E2 -17579.213} C_VEL
LIN {X 0,Y 286.475,Z 653.803,A -85,B 0,C 180,E1 -17581.423,E2 -17581.423} C_VEL
LIN {X 0,Y 288.372,Z 646.514,A -85,B 0,C 180,E1 -17583.257,E2 -17583.257} C_VEL
LIN {X 0,Y 290.495,Z 637.438,A -85,B 0,C 180,E1 -17585.096,E2 -17585.096} C_VEL
LIN {X 0,Y 292.4,Z 627.546,A -85,B 0,C 180,E1 -17586.721,E2 -17586.721} C_VEL
LIN {X 0,Y 294.375,Z 616.422,A -85,B 0,C 180,E1 -17588.147,E2 -17588.147} C_VEL
LIN {X 0,Y 295.868,Z 604.555,A -85,B 0,C 180,E1 -17589.343,E2 -17589.343} C_VEL
LIN {X 0,Y 296.912,Z 592.612,A -85,B 0,C 180,E1 -17590.262,E2 -17590.262} C_VEL
LIN {X 0,Y 297.535,Z 579.66,A -85,B 0,C 180,E1 -17590.97,E2 -17590.97} C_VEL
LIN {X 0,Y 297.79,Z 564.868,A -85,B 0,C 180,E1 -17591.457,E2 -17591.457} C_VEL
LIN {X 0,Y 298.629,Z 528.391,A -85,B 0,C 180,E1 -17592.396,E2 -17592.396} C_VEL
LIN {X 0,Y 291.256,Z 514.149,A -85,B 0,C 180,E1 -17593.811,E2 -17593.811} C_VEL
LIN {X 0,Y 286.266,Z 505.446,A -85,B 0,C 180,E1 -17594.801,E2 -17594.801} C_VEL
LIN {X 0,Y 284.673,Z 504.65,A -85,B 0,C 180,E1 -17595.065,E2 -17595.065} C_VEL
LIN {X 0,Y 282.191,Z 504.193,A -85,B 0,C 180,E1 -17595.459,E2 -17595.459} C_VEL
LIN {X 0,Y 280.693,Z 503.074,A -85,B 0,C 180,E1 -17595.827,E2 -17595.827} C_VEL
LIN {X 0,Y 280.442,Z 503.187,A -85,B 0,C 180,E1 -17596.207,E2 -17596.207} C_VEL
LIN {X 0,Y 283.12,Z 515.379,A -85,B 0,C 180,E1 -17599.099,E2 -17599.099} C_VEL
LIN {X 0,Y 283.755,Z 520.179,A -85,B 0,C 180,E1 -17600.16,E2 -17600.16} C_VEL
LIN {X 0,Y 283.28,Z 527.158,A -85,B 0,C 180,E1 -17601.583,E2 -17601.583} C_VEL
LIN {X 0,Y 286.745,Z 555.048,A -85,B 0,C 180,E1 -17602.81,E2 -17602.81} C_VEL
LIN {X 0,Y 284.413,Z 615.085,A -85,B 0,C 180,E1 -17604.813,E2 -17604.813} C_VEL
LIN {X 0,Y 283.617,Z 620.872,A -85,B 0,C 180,E1 -17604.978,E2 -17604.978} C_VEL
LIN {X 0,Y 277.374,Z 639.551,A -85,B 0,C 180,E1 -17605.429,E2 -17605.429} C_VEL
LIN {X 0,Y 276.345,Z 645.25,A -85,B 0,C 180,E1 -17605.683,E2 -17605.683} C_VEL
LIN {X 0,Y 275.502,Z 658.104,A -85,B 0,C 180,E1 -17606.52,E2 -17606.52} C_VEL
LIN {X 0,Y 274.572,Z 671.743,A -85,B 0,C 180,E1 -17607.743,E2 -17607.743} C_VEL
LIN {X 0,Y 273.466,Z 683.149,A -85,B 0,C 180,E1 -17609.07,E2 -17609.07} C_VEL
LIN {X 0,Y 272.346,Z 693.969,A -85,B 0,C 180,E1 -17610.64,E2 -17610.64} C_VEL
LIN {X 0,Y 271.467,Z 702.934,A -85,B 0,C 180,E1 -17612.226,E2 -17612.226} C_VEL
LIN {X 0,Y 270.502,Z 712.125,A -85,B 0,C 180,E1 -17614.203,E2 -17614.203} C_VEL
LIN {X 0,Y 269.723,Z 720.172,A -85,B 0,C 180,E1 -17616.337,E2 -17616.337} C_VEL
LIN {X 0,Y 269.048,Z 726.927,A -85,B 0,C 180,E1 -17618.55,E2 -17618.55} C_VEL
LIN {X 0,Y 268.639,Z 732.775,A -85,B 0,C 180,E1 -17621.001,E2 -17621.001} C_VEL
LIN {X 0,Y 268.328,Z 736.874,A -85,B 0,C 180,E1 -17623.256,E2 -17623.256} C_VEL
LIN {X 0,Y 268.254,Z 740.183,A -85,B 0,C 180,E1 -17625.789,E2 -17625.789} C_VEL
LIN {X 0,Y 268.306,Z 741.97,A -85,B 0,C 180,E1 -17627.904,E2 -17627.904} C_VEL
LIN {X 0,Y 268.454,Z 742.755,A -85,B 0,C 180,E1 -17629.441,E2 -17629.441} C_VEL
LIN {X 0,Y 268.723,Z 743.07,A -85,B 0,C 180,E1 -17630.972,E2 -17630.972} C_VEL
LIN {X 0,Y 269.19,Z 742.86,A -85,B 0,C 180,E1 -17632.81,E2 -17632.81} C_VEL
LIN {X 0,Y 270.076,Z 741.408,A -85,B 0,C 180,E1 -17635.523,E2 -17635.523} C_VEL
LIN {X 0,Y 270.753,Z 739.976,A -85,B 0,C 180,E1 -17637.025,E2 -17637.025} C_VEL
LIN {X 0,Y 272.06,Z 737.001,A -85,B 0,C 180,E1 -17639.26,E2 -17639.26} C_VEL
LIN {X 0,Y 273.705,Z 732.929,A -85,B 0,C 180,E1 -17641.472,E2 -17641.472} C_VEL
LIN {X 0,Y 276.052,Z 726.693,A -85,B 0,C 180,E1 -17644.015,E2 -17644.015} C_VEL
LIN {X 0,Y 278.424,Z 719.861,A -85,B 0,C 180,E1 -17646.159,E2 -17646.159} C_VEL
LIN {X 0,Y 281.198,Z 711.369,A -85,B 0,C 180,E1 -17648.263,E2 -17648.263} C_VEL
LIN {X 0,Y 283.715,Z 702.687,A -85,B 0,C 180,E1 -17649.986,E2 -17649.986} C_VEL
LIN {X 0,Y 286.231,Z 693.278,A -85,B 0,C 180,E1 -17651.508,E2 -17651.508} C_VEL
LIN {X 0,Y 288.867,Z 681.601,A -85,B 0,C 180,E1 -17653.043,E2 -17653.043} C_VEL
LIN {X 0,Y 291.14,Z 670.124,A -85,B 0,C 180,E1 -17654.194,E2 -17654.194} C_VEL
LIN {X 0,Y 293.015,Z 658.022,A -85,B 0,C 180,E1 -17655.148,E2 -17655.148} C_VEL
LIN {X 0,Y 294.568,Z 644.665,A -85,B 0,C 180,E1 -17655.925,E2 -17655.925} C_VEL
LIN {X 0,Y 302.134,Z 565.86,A -85,B 0,C 180,E1 -17658.903,E2 -17658.903} C_VEL
LIN {X 0,Y 300.444,Z 554.126,A -85,B 0,C 180,E1 -17660.075,E2 -17660.075} C_VEL
LIN {X 0,Y 297.394,Z 547.033,A -85,B 0,C 180,E1 -17661.396,E2 -17661.396} C_VEL
LIN {X 0,Y 293.376,Z 539.107,A -85,B 0,C 180,E1 -17663.249,E2 -17663.249} C_VEL
LIN {X 0,Y 291.187,Z 535.168,A -85,B 0,C 180,E1 -17664.415,E2 -17664.415} C_VEL
LIN {X 0,Y 290.268,Z 531,A -85,B 0,C 180,E1 -17666.378,E2 -17666.378} C_VEL
LIN {X 0,Y 289.029,Z 526.359,A -85,B 0,C 180,E1 -17669.099,E2 -17669.099} C_VEL
LIN {X 0,Y 288.143,Z 523.327,A -85,B 0,C 180,E1 -17671.383,E2 -17671.383} C_VEL
LIN {X 0,Y 287.261,Z 520.662,A -85,B 0,C 180,E1 -17674.244,E2 -17674.244} C_VEL
LIN {X 0,Y 286.985,Z 519.562,A -85,B 0,C 180,E1 -17676.082,E2 -17676.082} C_VEL
LIN {X 0,Y 287.032,Z 518.946,A -85,B 0,C 180,E1 -17679.54,E2 -17679.54} C_VEL
LIN {X 0,Y 287.441,Z 519.292,A -85,B 0,C 180,E1 -17681.312,E2 -17681.312} C_VEL
LIN {X 0,Y 288.132,Z 520.109,A -85,B 0,C 180,E1 -17683.076,E2 -17683.076} C_VEL
LIN {X 0,Y 289.443,Z 521.728,A -85,B 0,C 180,E1 -17685.236,E2 -17685.236} C_VEL
LIN {X 0,Y 290.417,Z 523.129,A -85,B 0,C 180,E1 -17686.552,E2 -17686.552} C_VEL
LIN {X 0,Y 291.316,Z 525.44,A -85,B 0,C 180,E1 -17687.889,E2 -17687.889} C_VEL
LIN {X 0,Y 292.287,Z 532.483,A -85,B 0,C 180,E1 -17690.304,E2 -17690.304} C_VEL
LIN {X 0,Y 293.87,Z 541.91,A -85,B 0,C 180,E1 -17692.868,E2 -17692.868} C_VEL
LIN {X 0,Y 294.757,Z 546.483,A -85,B 0,C 180,E1 -17693.935,E2 -17693.935} C_VEL
LIN {X 0,Y 296.31,Z 560.561,A -85,B 0,C 180,E1 -17695.42,E2 -17695.42} C_VEL
LIN {X 0,Y 297.571,Z 576.59,A -85,B 0,C 180,E1 -17696.814,E2 -17696.814} C_VEL
LIN {X 0,Y 298.19,Z 590.655,A -85,B 0,C 180,E1 -17697.868,E2 -17697.868} C_VEL
LIN {X 0,Y 298.119,Z 609.179,A -85,B 0,C 180,E1 -17698.95,E2 -17698.95} C_VEL
LIN {X 0,Y 292.4,Z 669.475,A -85,B 0,C 180,E1 -17701.266,E2 -17701.266} C_VEL
LIN {X 0,Y 290.403,Z 683.166,A -85,B 0,C 180,E1 -17702.035,E2 -17702.035} C_VEL
LIN {X 0,Y 287.777,Z 697.11,A -85,B 0,C 180,E1 -17703.138,E2 -17703.138} C_VEL
LIN {X 0,Y 285.001,Z 709.38,A -85,B 0,C 180,E1 -17704.432,E2 -17704.432} C_VEL
LIN {X 0,Y 281.96,Z 721.653,A -85,B 0,C 180,E1 -17706.104,E2 -17706.104} C_VEL
LIN {X 0,Y 279.125,Z 731.627,A -85,B 0,C 180,E1 -17707.808,E2 -17707.808} C_VEL
LIN {X 0,Y 276.285,Z 741.416,A -85,B 0,C 180,E1 -17709.913,E2 -17709.913} C_VEL
LIN {X 0,Y 273.792,Z 749.324,A -85,B 0,C 180,E1 -17712.057,E2 -17712.057} C_VEL
LIN {X 0,Y 272.069,Z 755.794,A -85,B 0,C 180,E1 -17714.26,E2 -17714.26} C_VEL
LIN {X 0,Y 270.411,Z 760.996,A -85,B 0,C 180,E1 -17716.47,E2 -17716.47} C_VEL
LIN {X 0,Y 269.411,Z 765.042,A -85,B 0,C 180,E1 -17718.715,E2 -17718.715} C_VEL
LIN {X 0,Y 268.725,Z 768.06,A -85,B 0,C 180,E1 -17720.969,E2 -17720.969} C_VEL
LIN {X 0,Y 268.455,Z 769.537,A -85,B 0,C 180,E1 -17722.476,E2 -17722.476} C_VEL
LIN {X 0,Y 268.362,Z 770.751,A -85,B 0,C 180,E1 -17724.367,E2 -17724.367} C_VEL
LIN {X 0,Y 268.425,Z 771.335,A -85,B 0,C 180,E1 -17726.996,E2 -17726.996} C_VEL
LIN {X 0,Y 268.539,Z 771.09,A -85,B 0,C 180,E1 -17728.498,E2 -17728.498} C_VEL
LIN {X 0,Y 268.843,Z 770.381,A -85,B 0,C 180,E1 -17729.997,E2 -17729.997} C_VEL
LIN {X 0,Y 268.735,Z 769.171,A -85,B 0,C 180,E1 -17731.496,E2 -17731.496} C_VEL
LIN {X 0,Y 268.57,Z 766.462,A -85,B 0,C 180,E1 -17733.748,E2 -17733.748} C_VEL
LIN {X 0,Y 268.626,Z 762.274,A -85,B 0,C 180,E1 -17736.177,E2 -17736.177} C_VEL
LIN {X 0,Y 268.764,Z 756.476,A -85,B 0,C 180,E1 -17738.645,E2 -17738.645} C_VEL
LIN {X 0,Y 269.121,Z 749.601,A -85,B 0,C 180,E1 -17740.911,E2 -17740.911} C_VEL
LIN {X 0,Y 269.834,Z 740.985,A -85,B 0,C 180,E1 -17743.171,E2 -17743.171} C_VEL
LIN {X 0,Y 270.712,Z 732.05,A -85,B 0,C 180,E1 -17745.044,E2 -17745.044} C_VEL
LIN {X 0,Y 271.75,Z 721.25,A -85,B 0,C 180,E1 -17746.882,E2 -17746.882} C_VEL
LIN {X 0,Y 272.951,Z 710.085,A -85,B 0,C 180,E1 -17748.383,E2 -17748.383} C_VEL
LIN {X 0,Y 273.983,Z 698.475,A -85,B 0,C 180,E1 -17749.671,E2 -17749.671} C_VEL
LIN {X 0,Y 275.542,Z 686.876,A -85,B 0,C 180,E1 -17751.114,E2 -17751.114} C_VEL
LIN {X 0,Y 277.001,Z 674.839,A -85,B 0,C 180,E1 -17752.268,E2 -17752.268} C_VEL
LIN {X 0,Y 278.14,Z 662.215,A -85,B 0,C 180,E1 -17753.153,E2 -17753.153} C_VEL
LIN {X 0,Y 278.974,Z 648.581,A -85,B 0,C 180,E1 -17753.796,E2 -17753.796} C_VEL
LIN {X 0,Y 279.989,Z 603.977,A -85,B 0,C 180,E1 -17754.967,E2 -17754.967} C_VEL
LIN {X 0,Y 274.179,Z 537.441,A -85,B 0,C 180,E1 -17757.251,E2 -17757.251} C_VEL
LIN {X 0,Y 275.936,Z 524.669,A -85,B 0,C 180,E1 -17760.191,E2 -17760.191} C_VEL
LIN {X 0,Y 276.462,Z 519.55,A -85,B 0,C 180,E1 -17761.405,E2 -17761.405} C_VEL
LIN {X 0,Y 273.914,Z 506.697,A -85,B 0,C 180,E1 -17764.809,E2 -17764.809} C_VEL
LIN {X 0,Y 270.998,Z 494.207,A -85,B 0,C 180,E1 -17768.326,E2 -17768.326} C_VEL
LIN {X 0,Y 270.209,Z 490.942,A -85,B 0,C 180,E1 -17769.335,E2 -17769.335} C_VEL
LIN {X 0,Y 270.141,Z 490.832,A -85,B 0,C 180,E1 -17773.243,E2 -17773.243} C_VEL
LIN {X 0,Y 270.163,Z 490.831,A -85,B 0,C 180,E1 -17777.439,E2 -17777.439} C_VEL
LIN {X 0,Y 270.198,Z 490.825,A -85,B 0,C 180,E1 -17781.372,E2 -17781.372} C_VEL
LIN {X 0,Y 270.188,Z 490.818,A -85,B 0,C 180,E1 -17785.092,E2 -17785.092} C_VEL
LIN {X 0,Y 270.19,Z 490.826,A -85,B 0,C 180,E1 -17789.129,E2 -17789.129} C_VEL
LIN {X 0,Y 270.253,Z 490.809,A -85,B 0,C 180,E1 -17792.144,E2 -17792.144} C_VEL
LIN {X 0,Y 270.266,Z 490.817,A -85,B 0,C 180,E1 -17795.518,E2 -17795.518} C_VEL
LIN {X 0,Y 270.29,Z 490.807,A -85,B 0,C 180,E1 -17800.243,E2 -17800.243} C_VEL
LIN {X 0,Y 270.391,Z 490.802,A -85,B 0,C 180,E1 -17804.934,E2 -17804.934} C_VEL
LIN {X 0,Y 270.429,Z 490.785,A -85,B 0,C 180,E1 -17809.518,E2 -17809.518} C_VEL
LIN {X 0,Y 270.598,Z 490.778,A -85,B 0,C 180,E1 -17812.538,E2 -17812.538} C_VEL
LIN {X 0,Y 270.774,Z 490.742,A -85,B 0,C 180,E1 -17818.512,E2 -17818.512} C_VEL
LIN {X 0,Y 270.775,Z 490.75,A -85,B 0,C 180,E1 -17821.487,E2 -17821.487} C_VEL
LIN {X 0,Y 270.597,Z 490.767,A -85,B 0,C 180,E1 -17827.461,E2 -17827.461} C_VEL
LIN {X 0,Y 270.428,Z 490.788,A -85,B 0,C 180,E1 -17830.481,E2 -17830.481} C_VEL
LIN {X 0,Y 270.389,Z 490.802,A -85,B 0,C 180,E1 -17835.065,E2 -17835.065} C_VEL
LIN {X 0,Y 270.288,Z 490.801,A -85,B 0,C 180,E1 -17839.756,E2 -17839.756} C_VEL
LIN {X 0,Y 270.261,Z 490.821,A -85,B 0,C 180,E1 -17844.586,E2 -17844.586} C_VEL
LIN {X 0,Y 270.259,Z 490.81,A -85,B 0,C 180,E1 -17847.909,E2 -17847.909} C_VEL
LIN {X 0,Y 270.172,Z 490.828,A -85,B 0,C 180,E1 -17851.349,E2 -17851.349} C_VEL
LIN {X 0,Y 270.189,Z 490.827,A -85,B 0,C 180,E1 -17854.907,E2 -17854.907} C_VEL
LIN {X 0,Y 270.185,Z 490.822,A -85,B 0,C 180,E1 -17858.712,E2 -17858.712} C_VEL
LIN {X 0,Y 270.177,Z 490.825,A -85,B 0,C 180,E1 -17863.256,E2 -17863.256} C_VEL
LIN {X 0,Y 270.238,Z 490.822,A -85,B 0,C 180,E1 -17867.458,E2 -17867.458} C_VEL
LIN {X 0,Y 270.235,Z 490.809,A -85,B 0,C 180,E1 -17871.382,E2 -17871.382} C_VEL
LIN {X 0,Y 270.207,Z 490.809,A -85,B 0,C 180,E1 -17875.099,E2 -17875.099} C_VEL
LIN {X 0,Y 270.192,Z 490.828,A -85,B 0,C 180,E1 -17879.133,E2 -17879.133} C_VEL
LIN {X 0,Y 270.256,Z 490.802,A -85,B 0,C 180,E1 -17882.148,E2 -17882.148} C_VEL
LIN {X 0,Y 270.27,Z 490.82,A -85,B 0,C 180,E1 -17885.521,E2 -17885.521} C_VEL
LIN {X 0,Y 270.296,Z 490.816,A -85,B 0,C 180,E1 -17890.247,E2 -17890.247} C_VEL
LIN {X 0,Y 270.398,Z 490.805,A -85,B 0,C 180,E1 -17894.938,E2 -17894.938} C_VEL
LIN {X 0,Y 270.42,Z 491.012,A -85,B 0,C 180,E1 -17897.269,E2 -17897.269} C_VEL
LIN {X 0,Y 270.66,Z 491.974,A -85,B 0,C 180,E1 -17897.506,E2 -17897.506} C_VEL
LIN {X 0,Y 279.962,Z 513.893,A -85,B 0,C 180,E1 -17898.925,E2 -17898.925} C_VEL
LIN {X 0,Y 281.495,Z 518.267,A -85,B 0,C 180,E1 -17899.166,E2 -17899.166} C_VEL
LIN {X 0,Y 280.553,Z 561.336,A -85,B 0,C 180,E1 -17900.261,E2 -17900.261} C_VEL
LIN {X 0,Y 280.434,Z 578.587,A -85,B 0,C 180,E1 -17900.815,E2 -17900.815} C_VEL
LIN {X 0,Y 280.013,Z 591.373,A -85,B 0,C 180,E1 -17901.523,E2 -17901.523} C_VEL
LIN {X 0,Y 279.284,Z 604.687,A -85,B 0,C 180,E1 -17902.593,E2 -17902.593} C_VEL
LIN {X 0,Y 278.307,Z 616.387,A -85,B 0,C 180,E1 -17903.841,E2 -17903.841} C_VEL
LIN {X 0,Y 277.027,Z 628.064,A -85,B 0,C 180,E1 -17905.455,E2 -17905.455} C_VEL
LIN {X 0,Y 275.932,Z 637.465,A -85,B 0,C 180,E1 -17907.083,E2 -17907.083} C_VEL
LIN {X 0,Y 274.698,Z 646.496,A -85,B 0,C 180,E1 -17908.998,E2 -17908.998} C_VEL
LIN {X 0,Y 273.54,Z 654.47,A -85,B 0,C 180,E1 -17911.107,E2 -17911.107} C_VEL
LIN {X 0,Y 272.54,Z 661.227,A -85,B 0,C 180,E1 -17913.329,E2 -17913.329} C_VEL
LIN {X 0,Y 271.673,Z 667.449,A -85,B 0,C 180,E1 -17915.942,E2 -17915.942} C_VEL
LIN {X 0,Y 271.126,Z 671.517,A -85,B 0,C 180,E1 -17918.199,E2 -17918.199} C_VEL
LIN {X 0,Y 270.757,Z 674.553,A -85,B 0,C 180,E1 -17920.471,E2 -17920.471} C_VEL
LIN {X 0,Y 270.667,Z 676.01,A -85,B 0,C 180,E1 -17921.991,E2 -17921.991} C_VEL
LIN {X 0,Y 270.805,Z 677.728,A -85,B 0,C 180,E1 -17925.044,E2 -17925.044} C_VEL
LIN {X 0,Y 271.035,Z 677.976,A -85,B 0,C 180,E1 -17926.575,E2 -17926.575} C_VEL
LIN {X 0,Y 271.362,Z 677.793,A -85,B 0,C 180,E1 -17928.109,E2 -17928.109} C_VEL
LIN {X 0,Y 271.771,Z 677.22,A -85,B 0,C 180,E1 -17929.647,E2 -17929.647} C_VEL
LIN {X 0,Y 272.658,Z 675.603,A -85,B 0,C 180,E1 -17931.887,E2 -17931.887} C_VEL
LIN {X 0,Y 274.302,Z 671.752,A -85,B 0,C 180,E1 -17935.011,E2 -17935.011} C_VEL
LIN {X 0,Y 275.846,Z 667.594,A -85,B 0,C 180,E1 -17937.3,E2 -17937.3} C_VEL
LIN {X 0,Y 277.688,Z 662.161,A -85,B 0,C 180,E1 -17939.575,E2 -17939.575} C_VEL
LIN {X 0,Y 279.838,Z 655.255,A -85,B 0,C 180,E1 -17941.833,E2 -17941.833} C_VEL
LIN {X 0,Y 281.8,Z 648.085,A -85,B 0,C 180,E1 -17943.707,E2 -17943.707} C_VEL
LIN {X 0,Y 284.009,Z 639.222,A -85,B 0,C 180,E1 -17945.566,E2 -17945.566} C_VEL
LIN {X 0,Y 286.033,Z 629.397,A -85,B 0,C 180,E1 -17947.235,E2 -17947.235} C_VEL
LIN {X 0,Y 288.055,Z 618.663,A -85,B 0,C 180,E1 -17948.673,E2 -17948.673} C_VEL
LIN {X 0,Y 289.643,Z 607.01,A -85,B 0,C 180,E1 -17949.906,E2 -17949.906} C_VEL
LIN {X 0,Y 290.871,Z 594.158,A -85,B 0,C 180,E1 -17950.933,E2 -17950.933} C_VEL
LIN {X 0,Y 291.55,Z 581.731,A -85,B 0,C 180,E1 -17951.646,E2 -17951.646} C_VEL
LIN {X 0,Y 291.816,Z 568.16,A -85,B 0,C 180,E1 -17952.128,E2 -17952.128} C_VEL
LIN {X 0,Y 292.726,Z 530.655,A -85,B 0,C 180,E1 -17953.113,E2 -17953.113} C_VEL
LIN {X 0,Y 284.332,Z 514.667,A -85,B 0,C 180,E1 -17954.803,E2 -17954.803} C_VEL
LIN {X 0,Y 282.382,Z 511.546,A -85,B 0,C 180,E1 -17955.197,E2 -17955.197} C_VEL
LIN {X 0,Y 279.287,Z 510.553,A -85,B 0,C 180,E1 -17955.71,E2 -17955.71} C_VEL
LIN {X 0,Y 277.904,Z 510.315,A -85,B 0,C 180,E1 -17955.937,E2 -17955.937} C_VEL
LIN {X 0,Y 275.712,Z 509.646,A -85,B 0,C 180,E1 -17956.321,E2 -17956.321} C_VEL
LIN {X 0,Y 274.636,Z 508.776,A -85,B 0,C 180,E1 -17956.674,E2 -17956.674} C_VEL
LIN {X 0,Y 274.526,Z 509.083,A -85,B 0,C 180,E1 -17957.014,E2 -17957.014} C_VEL
LIN {X 0,Y 276.823,Z 519.974,A -85,B 0,C 180,E1 -17959.612,E2 -17959.612} C_VEL
LIN {X 0,Y 276.466,Z 527.52,A -85,B 0,C 180,E1 -17961.173,E2 -17961.173} C_VEL
LIN {X 0,Y 279.901,Z 555.473,A -85,B 0,C 180,E1 -17962.439,E2 -17962.439} C_VEL
LIN {X 0,Y 276.558,Z 639.683,A -85,B 0,C 180,E1 -17965.403,E2 -17965.403} C_VEL
LIN {X 0,Y 276.345,Z 645.25,A -85,B 0,C 180,E1 -17965.683,E2 -17965.683} C_VEL
LIN {X 0,Y 275.262,Z 650.894,A -85,B 0,C 180,E1 -17965.976,E2 -17965.976} C_VEL
LIN {X 0,Y 271.91,Z 659.877,A -85,B 0,C 180,E1 -17966.506,E2 -17966.506} C_VEL
LIN {X 0,Y 268.516,Z 668.602,A -85,B 0,C 180,E1 -17967.191,E2 -17967.191} C_VEL
LIN {X 0,Y 267.375,Z 673.84,A -85,B 0,C 180,E1 -17967.722,E2 -17967.722} C_VEL
LIN {X 0,Y 266.203,Z 686.028,A -85,B 0,C 180,E1 -17969.236,E2 -17969.236} C_VEL
LIN {X 0,Y 265.058,Z 696.784,A -85,B 0,C 180,E1 -17970.917,E2 -17970.917} C_VEL
LIN {X 0,Y 264.1,Z 705.973,A -85,B 0,C 180,E1 -17972.675,E2 -17972.675} C_VEL
LIN {X 0,Y 263.204,Z 714.703,A -85,B 0,C 180,E1 -17974.709,E2 -17974.709} C_VEL
LIN {X 0,Y 262.474,Z 721.83,A -85,B 0,C 180,E1 -17976.738,E2 -17976.738} C_VEL
LIN {X 0,Y 261.824,Z 728.673,A -85,B 0,C 180,E1 -17979.167,E2 -17979.167} C_VEL
LIN {X 0,Y 261.498,Z 733.239,A -85,B 0,C 180,E1 -17981.186,E2 -17981.186} C_VEL
LIN {X 0,Y 261.208,Z 737.472,A -85,B 0,C 180,E1 -17983.591,E2 -17983.591} C_VEL
LIN {X 0,Y 261.16,Z 740.528,A -85,B 0,C 180,E1 -17985.984,E2 -17985.984} C_VEL
LIN {X 0,Y 261.209,Z 741.978,A -85,B 0,C 180,E1 -17987.571,E2 -17987.571} C_VEL
LIN {X 0,Y 261.317,Z 742.925,A -85,B 0,C 180,E1 -17989.149,E2 -17989.149} C_VEL
LIN {X 0,Y 261.595,Z 743.436,A -85,B 0,C 180,E1 -17990.724,E2 -17990.724} C_VEL
LIN {X 0,Y 262.11,Z 743.44,A -85,B 0,C 180,E1 -17992.803,E2 -17992.803} C_VEL
LIN {X 0,Y 262.966,Z 742.365,A -85,B 0,C 180,E1 -17995.402,E2 -17995.402} C_VEL
LIN {X 0,Y 263.65,Z 741.164,A -85,B 0,C 180,E1 -17996.944,E2 -17996.944} C_VEL
LIN {X 0,Y 264.983,Z 738.494,A -85,B 0,C 180,E1 -17999.241,E2 -17999.241} C_VEL
LIN {X 0,Y 266.675,Z 734.792,A -85,B 0,C 180,E1 -18001.511,E2 -18001.511} C_VEL
LIN {X 0,Y 268.687,Z 729.954,A -85,B 0,C 180,E1 -18003.75,E2 -18003.75} C_VEL
LIN {X 0,Y 271.129,Z 723.768,A -85,B 0,C 180,E1 -18005.952,E2 -18005.952} C_VEL
LIN {X 0,Y 273.865,Z 716.112,A -85,B 0,C 180,E1 -18008.115,E2 -18008.115} C_VEL
LIN {X 0,Y 276.469,Z 708.385,A -85,B 0,C 180,E1 -18009.881,E2 -18009.881} C_VEL
LIN {X 0,Y 279.25,Z 699.052,A -85,B 0,C 180,E1 -18011.616,E2 -18011.616} C_VEL
LIN {X 0,Y 282.078,Z 688.285,A -85,B 0,C 180,E1 -18013.209,E2 -18013.209} C_VEL
LIN {X 0,Y 284.533,Z 677.595,A -85,B 0,C 180,E1 -18014.483,E2 -18014.483} C_VEL
LIN {X 0,Y 286.923,Z 665.192,A -85,B 0,C 180,E1 -18015.631,E2 -18015.631} C_VEL
LIN {X 0,Y 288.856,Z 651.94,A -85,B 0,C 180,E1 -18016.567,E2 -18016.567} C_VEL
LIN {X 0,Y 290.497,Z 636.54,A -85,B 0,C 180,E1 -18017.285,E2 -18017.285} C_VEL
LIN {X 0,Y 297.627,Z 567.741,A -85,B 0,C 180,E1 -18019.91,E2 -18019.91} C_VEL
LIN {X 0,Y 296.296,Z 558.062,A -85,B 0,C 180,E1 -18020.919,E2 -18020.919} C_VEL
LIN {X 0,Y 293.699,Z 551.782,A -85,B 0,C 180,E1 -18022.153,E2 -18022.153} C_VEL
LIN {X 0,Y 290.343,Z 544.799,A -85,B 0,C 180,E1 -18023.84,E2 -18023.84} C_VEL
LIN {X 0,Y 287.02,Z 538.978,A -85,B 0,C 180,E1 -18025.67,E2 -18025.67} C_VEL
LIN {X 0,Y 285.583,Z 536.089,A -85,B 0,C 180,E1 -18026.688,E2 -18026.688} C_VEL
LIN {X 0,Y 284.455,Z 531.344,A -85,B 0,C 180,E1 -18029.613,E2 -18029.613} C_VEL
LIN {X 0,Y 283.921,Z 529.177,A -85,B 0,C 180,E1 -18031.321,E2 -18031.321} C_VEL
LIN {X 0,Y 283.097,Z 526.078,A -85,B 0,C 180,E1 -18034.988,E2 -18034.988} C_VEL
LIN {X 0,Y 282.961,Z 525.131,A -85,B 0,C 180,E1 -18037.361,E2 -18037.361} C_VEL
LIN {X 0,Y 283.393,Z 525.054,A -85,B 0,C 180,E1 -18040.15,E2 -18040.15} C_VEL
LIN {X 0,Y 284.009,Z 525.683,A -85,B 0,C 180,E1 -18042.063,E2 -18042.063} C_VEL
LIN {X 0,Y 285.974,Z 528.104,A -85,B 0,C 180,E1 -18045.455,E2 -18045.455} C_VEL
LIN {X 0,Y 287.267,Z 530.421,A -85,B 0,C 180,E1 -18047.219,E2 -18047.219} C_VEL
LIN {X 0,Y 287.959,Z 535.695,A -85,B 0,C 180,E1 -18049.166,E2 -18049.166} C_VEL
LIN {X 0,Y 289.136,Z 544.428,A -85,B 0,C 180,E1 -18051.711,E2 -18051.711} C_VEL
LIN {X 0,Y 290.396,Z 548.599,A -85,B 0,C 180,E1 -18052.655,E2 -18052.655} C_VEL
LIN {X 0,Y 291.15,Z 551.244,A -85,B 0,C 180,E1 -18053.136,E2 -18053.136} C_VEL
LIN {X 0,Y 292.59,Z 567.991,A -85,B 0,C 180,E1 -18054.87,E2 -18054.87} C_VEL
LIN {X 0,Y 293.535,Z 586.256,A -85,B 0,C 180,E1 -18056.422,E2 -18056.422} C_VEL
LIN {X 0,Y 293.622,Z 600.208,A -85,B 0,C 180,E1 -18057.365,E2 -18057.365} C_VEL
LIN {X 0,Y 293.212,Z 611.914,A -85,B 0,C 180,E1 -18058.021,E2 -18058.021} C_VEL
LIN {X 0,Y 287.516,Z 668.426,A -85,B 0,C 180,E1 -18060.228,E2 -18060.228} C_VEL
LIN {X 0,Y 285.399,Z 682.054,A -85,B 0,C 180,E1 -18060.998,E2 -18060.998} C_VEL
LIN {X 0,Y 282.804,Z 695.048,A -85,B 0,C 180,E1 -18062.024,E2 -18062.024} C_VEL
LIN {X 0,Y 280.173,Z 706.3,A -85,B 0,C 180,E1 -18063.156,E2 -18063.156} C_VEL
LIN {X 0,Y 277.17,Z 717.873,A -85,B 0,C 180,E1 -18064.664,E2 -18064.664} C_VEL
LIN {X 0,Y 273.793,Z 729.331,A -85,B 0,C 180,E1 -18066.552,E2 -18066.552} C_VEL
LIN {X 0,Y 270.625,Z 739.378,A -85,B 0,C 180,E1 -18068.678,E2 -18068.678} C_VEL
LIN {X 0,Y 268.204,Z 746.796,A -85,B 0,C 180,E1 -18070.622,E2 -18070.622} C_VEL
LIN {X 0,Y 266.101,Z 753.255,A -85,B 0,C 180,E1 -18072.713,E2 -18072.713} C_VEL
LIN {X 0,Y 264.07,Z 759.658,A -85,B 0,C 180,E1 -18075.352,E2 -18075.352} C_VEL
LIN {X 0,Y 262.724,Z 763.914,A -85,B 0,C 180,E1 -18077.64,E2 -18077.64} C_VEL
LIN {X 0,Y 262.126,Z 766.144,A -85,B 0,C 180,E1 -18079.18,E2 -18079.18} C_VEL
LIN {X 0,Y 261.696,Z 767.954,A -85,B 0,C 180,E1 -18080.725,E2 -18080.725} C_VEL
LIN {X 0,Y 261.38,Z 769.323,A -85,B 0,C 180,E1 -18082.271,E2 -18082.271} C_VEL
LIN {X 0,Y 261.267,Z 770.525,A -85,B 0,C 180,E1 -18084.441,E2 -18084.441} C_VEL
LIN {X 0,Y 261.349,Z 770.872,A -85,B 0,C 180,E1 -18086.914,E2 -18086.914} C_VEL
LIN {X 0,Y 261.457,Z 770.507,A -85,B 0,C 180,E1 -18088.457,E2 -18088.457} C_VEL
LIN {X 0,Y 261.783,Z 769.713,A -85,B 0,C 180,E1 -18089.997,E2 -18089.997} C_VEL
LIN {X 0,Y 261.664,Z 768.441,A -85,B 0,C 180,E1 -18091.536,E2 -18091.536} C_VEL
LIN {X 0,Y 261.509,Z 765.607,A -85,B 0,C 180,E1 -18093.85,E2 -18093.85} C_VEL
LIN {X 0,Y 261.569,Z 761.549,A -85,B 0,C 180,E1 -18096.202,E2 -18096.202} C_VEL
LIN {X 0,Y 261.738,Z 755.241,A -85,B 0,C 180,E1 -18098.879,E2 -18098.879} C_VEL
LIN {X 0,Y 262.112,Z 748.175,A -85,B 0,C 180,E1 -18101.207,E2 -18101.207} C_VEL
LIN {X 0,Y 262.724,Z 740.9,A -85,B 0,C 180,E1 -18103.14,E2 -18103.14} C_VEL
LIN {X 0,Y 263.61,Z 732.03,A -85,B 0,C 180,E1 -18105.064,E2 -18105.064} C_VEL
LIN {X 0,Y 264.677,Z 721.121,A -85,B 0,C 180,E1 -18106.98,E2 -18106.98} C_VEL
LIN {X 0,Y 265.859,Z 710.267,A -85,B 0,C 180,E1 -18108.492,E2 -18108.492} C_VEL
LIN {X 0,Y 266.888,Z 699.168,A -85,B 0,C 180,E1 -18109.815,E2 -18109.815} C_VEL
LIN {X 0,Y 268.425,Z 688.019,A -85,B 0,C 180,E1 -18111.299,E2 -18111.299} C_VEL
LIN {X 0,Y 269.596,Z 679.529,A -85,B 0,C 180,E1 -18112.207,E2 -18112.207} C_VEL
LIN {X 0,Y 270.904,Z 667.662,A -85,B 0,C 180,E1 -18113.201,E2 -18113.201} C_VEL
LIN {X 0,Y 271.944,Z 653.94,A -85,B 0,C 180,E1 -18114.016,E2 -18114.016} C_VEL
LIN {X 0,Y 272.562,Z 640.442,A -85,B 0,C 180,E1 -18114.504,E2 -18114.504} C_VEL
LIN {X 0,Y 273.237,Z 603.661,A -85,B 0,C 180,E1 -18115.471,E2 -18115.471} C_VEL
LIN {X 0,Y 267.382,Z 536.554,A -85,B 0,C 180,E1 -18117.837,E2 -18117.837} C_VEL
LIN {X 0,Y 267.818,Z 533.031,A -85,B 0,C 180,E1 -18118.611,E2 -18118.611} C_VEL
LIN {X 0,Y 269.494,Z 521.357,A -85,B 0,C 180,E1 -18121.434,E2 -18121.434} C_VEL
LIN {X 0,Y 267.479,Z 510.422,A -85,B 0,C 180,E1 -18124.393,E2 -18124.393} C_VEL
LIN {X 0,Y 264.704,Z 498.079,A -85,B 0,C 180,E1 -18127.922,E2 -18127.922} C_VEL
LIN {X 0,Y 263.124,Z 491.82,A -85,B 0,C 180,E1 -18129.865,E2 -18129.865} C_VEL
LIN {X 0,Y 263.09,Z 491.711,A -85,B 0,C 180,E1 -18133.987,E2 -18133.987} C_VEL
LIN {X 0,Y 263.116,Z 491.712,A -85,B 0,C 180,E1 -18138.404,E2 -18138.404} C_VEL
LIN {X 0,Y 263.147,Z 491.707,A -85,B 0,C 180,E1 -18142.1,E2 -18142.1} C_VEL
LIN {X 0,Y 263.141,Z 491.697,A -85,B 0,C 180,E1 -18145.883,E2 -18145.883} C_VEL
LIN {X 0,Y 263.131,Z 491.706,A -85,B 0,C 180,E1 -18149.504,E2 -18149.504} C_VEL
LIN {X 0,Y 263.181,Z 491.694,A -85,B 0,C 180,E1 -18153.001,E2 -18153.001} C_VEL
LIN {X 0,Y 263.173,Z 491.705,A -85,B 0,C 180,E1 -18156.385,E2 -18156.385} C_VEL
LIN {X 0,Y 263.252,Z 491.684,A -85,B 0,C 180,E1 -18159.692,E2 -18159.692} C_VEL
LIN {X 0,Y 263.339,Z 491.684,A -85,B 0,C 180,E1 -18164.521,E2 -18164.521} C_VEL
LIN {X 0,Y 263.361,Z 491.665,A -85,B 0,C 180,E1 -18169.233,E2 -18169.233} C_VEL
LIN {X 0,Y 263.559,Z 491.653,A -85,B 0,C 180,E1 -18172.337,E2 -18172.337} C_VEL
LIN {X 0,Y 263.738,Z 491.617,A -85,B 0,C 180,E1 -18178.472,E2 -18178.472} C_VEL
LIN {X 0,Y 263.739,Z 491.626,A -85,B 0,C 180,E1 -18181.526,E2 -18181.526} C_VEL
LIN {X 0,Y 263.559,Z 491.642,A -85,B 0,C 180,E1 -18187.661,E2 -18187.661} C_VEL
LIN {X 0,Y 263.361,Z 491.67,A -85,B 0,C 180,E1 -18190.766,E2 -18190.766} C_VEL
LIN {X 0,Y 263.338,Z 491.679,A -85,B 0,C 180,E1 -18195.478,E2 -18195.478} C_VEL
LIN {X 0,Y 263.25,Z 491.678,A -85,B 0,C 180,E1 -18200.307,E2 -18200.307} C_VEL
LIN {X 0,Y 263.196,Z 491.697,A -85,B 0,C 180,E1 -18205.292,E2 -18205.292} C_VEL
LIN {X 0,Y 263.167,Z 491.691,A -85,B 0,C 180,E1 -18208.73,E2 -18208.73} C_VEL
LIN {X 0,Y 263.12,Z 491.707,A -85,B 0,C 180,E1 -18212.289,E2 -18212.289} C_VEL
LIN {X 0,Y 263.169,Z 491.694,A -85,B 0,C 180,E1 -18216.764,E2 -18216.764} C_VEL
LIN {X 0,Y 263.118,Z 491.708,A -85,B 0,C 180,E1 -18221.596,E2 -18221.596} C_VEL
LIN {X 0,Y 263.134,Z 491.702,A -85,B 0,C 180,E1 -18226.022,E2 -18226.022} C_VEL
LIN {X 0,Y 263.2,Z 491.699,A -85,B 0,C 180,E1 -18228.387,E2 -18228.387} C_VEL
LIN {X 0,Y 263.197,Z 491.671,A -85,B 0,C 180,E1 -18233.232,E2 -18233.232} C_VEL
LIN {X 0,Y 263.175,Z 491.694,A -85,B 0,C 180,E1 -18235.892,E2 -18235.892} C_VEL
LIN {X 0,Y 263.14,Z 491.704,A -85,B 0,C 180,E1 -18239.509,E2 -18239.509} C_VEL
LIN {X 0,Y 263.185,Z 491.685,A -85,B 0,C 180,E1 -18243.005,E2 -18243.005} C_VEL
LIN {X 0,Y 263.178,Z 491.703,A -85,B 0,C 180,E1 -18246.389,E2 -18246.389} C_VEL
LIN {X 0,Y 263.258,Z 491.688,A -85,B 0,C 180,E1 -18249.696,E2 -18249.696} C_VEL
LIN {X 0,Y 263.346,Z 491.681,A -85,B 0,C 180,E1 -18254.525,E2 -18254.525} C_VEL
LIN {X 0,Y 263.368,Z 491.893,A -85,B 0,C 180,E1 -18256.637,E2 -18256.637} C_VEL
LIN {X 0,Y 263.587,Z 492.796,A -85,B 0,C 180,E1 -18256.876,E2 -18256.876} C_VEL
LIN {X 0,Y 273.091,Z 514.898,A -85,B 0,C 180,E1 -18258.387,E2 -18258.387} C_VEL
LIN {X 0,Y 274.869,Z 519.613,A -85,B 0,C 180,E1 -18258.668,E2 -18258.668} C_VEL
LIN {X 0,Y 273.907,Z 560.809,A -85,B 0,C 180,E1 -18259.737,E2 -18259.737} C_VEL
LIN {X 0,Y 273.751,Z 578.638,A -85,B 0,C 180,E1 -18260.306,E2 -18260.306} C_VEL
LIN {X 0,Y 273.381,Z 590.873,A -85,B 0,C 180,E1 -18260.97,E2 -18260.97} C_VEL
LIN {X 0,Y 272.813,Z 602.332,A -85,B 0,C 180,E1 -18261.857,E2 -18261.857} C_VEL
LIN {X 0,Y 271.798,Z 614.731,A -85,B 0,C 180,E1 -18263.134,E2 -18263.134} C_VEL
LIN {X 0,Y 270.62,Z 625.825,A -85,B 0,C 180,E1 -18264.601,E2 -18264.601} C_VEL
LIN {X 0,Y 269.374,Z 635.844,A -85,B 0,C 180,E1 -18266.263,E2 -18266.263} C_VEL
LIN {X 0,Y 268.141,Z 644.887,A -85,B 0,C 180,E1 -18268.125,E2 -18268.125} C_VEL
LIN {X 0,Y 266.833,Z 653.727,A -85,B 0,C 180,E1 -18270.38,E2 -18270.38} C_VEL
LIN {X 0,Y 265.771,Z 660.842,A -85,B 0,C 180,E1 -18272.655,E2 -18272.655} C_VEL
LIN {X 0,Y 264.81,Z 667.338,A -85,B 0,C 180,E1 -18275.332,E2 -18275.332} C_VEL
LIN {X 0,Y 264.213,Z 671.652,A -85,B 0,C 180,E1 -18277.645,E2 -18277.645} C_VEL
LIN {X 0,Y 263.824,Z 674.618,A -85,B 0,C 180,E1 -18279.724,E2 -18279.724} C_VEL
LIN {X 0,Y 263.624,Z 677.194,A -85,B 0,C 180,E1 -18282.317,E2 -18282.317} C_VEL
LIN {X 0,Y 263.685,Z 678.194,A -85,B 0,C 180,E1 -18283.882,E2 -18283.882} C_VEL
LIN {X 0,Y 264.013,Z 678.969,A -85,B 0,C 180,E1 -18286.604,E2 -18286.604} C_VEL
LIN {X 0,Y 264.46,Z 678.721,A -85,B 0,C 180,E1 -18288.599,E2 -18288.599} C_VEL
LIN {X 0,Y 264.944,Z 678.094,A -85,B 0,C 180,E1 -18290.175,E2 -18290.175} C_VEL
LIN {X 0,Y 265.808,Z 676.55,A -85,B 0,C 180,E1 -18292.272,E2 -18292.272} C_VEL
LIN {X 0,Y 267.21,Z 673.535,A -85,B 0,C 180,E1 -18294.889,E2 -18294.889} C_VEL
LIN {X 0,Y 268.777,Z 669.629,A -85,B 0,C 180,E1 -18297.249,E2 -18297.249} C_VEL
LIN {X 0,Y 270.98,Z 663.514,A -85,B 0,C 180,E1 -18299.954,E2 -18299.954} C_VEL
LIN {X 0,Y 272.992,Z 657.364,A -85,B 0,C 180,E1 -18302.057,E2 -18302.057} C_VEL
LIN {X 0,Y 275.246,Z 649.622,A -85,B 0,C 180,E1 -18304.179,E2 -18304.179} C_VEL
LIN {X 0,Y 277.467,Z 641.321,A -85,B 0,C 180,E1 -18305.996,E2 -18305.996} C_VEL
LIN {X 0,Y 279.691,Z 631.248,A -85,B 0,C 180,E1 -18307.772,E2 -18307.772} C_VEL
LIN {X 0,Y 281.601,Z 621.499,A -85,B 0,C 180,E1 -18309.143,E2 -18309.143} C_VEL
LIN {X 0,Y 283.335,Z 610.391,A -85,B 0,C 180,E1 -18310.395,E2 -18310.395} C_VEL
LIN {X 0,Y 284.631,Z 598.248,A -85,B 0,C 180,E1 -18311.459,E2 -18311.459} C_VEL
LIN {X 0,Y 285.554,Z 584.78,A -85,B 0,C 180,E1 -18312.295,E2 -18312.295} C_VEL
LIN {X 0,Y 285.87,Z 573.369,A -85,B 0,C 180,E1 -18312.768,E2 -18312.768} C_VEL
LIN {X 0,Y 286.843,Z 536.47,A -85,B 0,C 180,E1 -18313.761,E2 -18313.761} C_VEL
LIN {X 0,Y 286.843,Z 532.959,A -85,B 0,C 180,E1 -18313.868,E2 -18313.868} C_VEL
LIN {X 0,Y 278.964,Z 518.057,A -85,B 0,C 180,E1 -18315.519,E2 -18315.519} C_VEL
LIN {X 0,Y 277.266,Z 517.379,A -85,B 0,C 180,E1 -18315.809,E2 -18315.809} C_VEL
LIN {X 0,Y 273.809,Z 516.587,A -85,B 0,C 180,E1 -18316.399,E2 -18316.399} C_VEL
LIN {X 0,Y 273.114,Z 516.194,A -85,B 0,C 180,E1 -18316.528,E2 -18316.528} C_VEL
LIN {X 0,Y 269.973,Z 515.62,A -85,B 0,C 180,E1 -18317.085,E2 -18317.085} C_VEL
LIN {X 0,Y 268.833,Z 514.716,A -85,B 0,C 180,E1 -18317.428,E2 -18317.428} C_VEL
LIN {X 0,Y 268.651,Z 514.931,A -85,B 0,C 180,E1 -18317.812,E2 -18317.812} C_VEL
LIN {X 0,Y 269.973,Z 522.448,A -85,B 0,C 180,E1 -18319.644,E2 -18319.644} C_VEL
LIN {X 0,Y 269.597,Z 528.006,A -85,B 0,C 180,E1 -18320.779,E2 -18320.779} C_VEL
LIN {X 0,Y 272.984,Z 556.502,A -85,B 0,C 180,E1 -18322.097,E2 -18322.097} C_VEL
LIN {X 0,Y 269.592,Z 639.737,A -85,B 0,C 180,E1 -18325.119,E2 -18325.119} C_VEL
LIN {X 0,Y 268.974,Z 652.198,A -85,B 0,C 180,E1 -18325.822,E2 -18325.822} C_VEL
LIN {X 0,Y 267.987,Z 665.963,A -85,B 0,C 180,E1 -18326.924,E2 -18326.924} C_VEL
LIN {X 0,Y 267.375,Z 673.84,A -85,B 0,C 180,E1 -18327.722,E2 -18327.722} C_VEL
LIN {X 0,Y 266.171,Z 679.074,A -85,B 0,C 180,E1 -18328.302,E2 -18328.302} C_VEL
LIN {X 0,Y 262.494,Z 687.175,A -85,B 0,C 180,E1 -18329.284,E2 -18329.284} C_VEL
LIN {X 0,Y 258.882,Z 694.776,A -85,B 0,C 180,E1 -18330.41,E2 -18330.41} C_VEL
LIN {X 0,Y 257.777,Z 699.276,A -85,B 0,C 180,E1 -18331.198,E2 -18331.198} C_VEL
LIN {X 0,Y 256.729,Z 708.744,A -85,B 0,C 180,E1 -18333.149,E2 -18333.149} C_VEL
LIN {X 0,Y 255.865,Z 717.243,A -85,B 0,C 180,E1 -18335.304,E2 -18335.304} C_VEL
LIN {X 0,Y 255.088,Z 725.033,A -85,B 0,C 180,E1 -18337.739,E2 -18337.739} C_VEL
LIN {X 0,Y 254.646,Z 730.296,A -85,B 0,C 180,E1 -18339.786,E2 -18339.786} C_VEL
LIN {X 0,Y 254.23,Z 735.433,A -85,B 0,C 180,E1 -18342.297,E2 -18342.297} C_VEL
LIN {X 0,Y 254.066,Z 739.314,A -85,B 0,C 180,E1 -18344.847,E2 -18344.847} C_VEL
LIN {X 0,Y 254.083,Z 741.837,A -85,B 0,C 180,E1 -18347.216,E2 -18347.216} C_VEL
